LIN {X 0,Y 474.649,Z 278.987,A -85,B 0,C 180,E1 -7371.485,E2 -7371.485} C_VEL
LIN {X 0,Y 474.743,Z 278.967,A -85,B 0,C 180,E1 -7374.052,E2 -7374.052} C_VEL
LIN {X 0,Y 474.863,Z 278.959,A -85,B 0,C 180,E1 -7377.455,E2 -7377.455} C_VEL
LIN {X 0,Y 474.863,Z 278.956,A -85,B 0,C 180,E1 -7380,E2 -7380} C_VEL
LIN {X 0,Y 474.868,Z 278.952,A -85,B 0,C 180,E1 -7382.545,E2 -7382.545} C_VEL
LIN {X 0,Y 474.745,Z 278.969,A -85,B 0,C 180,E1 -7385.948,E2 -7385.948} C_VEL
LIN {X 0,Y 474.696,Z 278.976,A -85,B 0,C 180,E1 -7388.514,E2 -7388.514} C_VEL
LIN {X 0,Y 474.691,Z 278.977,A -85,B 0,C 180,E1 -7391.963,E2 -7391.963} C_VEL
LIN {X 0,Y 474.667,Z 278.98,A -85,B 0,C 180,E1 -7395.767,E2 -7395.767} C_VEL
LIN {X 0,Y 474.65,Z 278.981,A -85,B 0,C 180,E1 -7399.011,E2 -7399.011} C_VEL
LIN {X 0,Y 474.576,Z 278.987,A -85,B 0,C 180,E1 -7401.73,E2 -7401.73} C_VEL
LIN {X 0,Y 474.618,Z 278.988,A -85,B 0,C 180,E1 -7404.495,E2 -7404.495} C_VEL
LIN {X 0,Y 474.663,Z 278.974,A -85,B 0,C 180,E1 -7407.333,E2 -7407.333} C_VEL
LIN {X 0,Y 474.594,Z 278.989,A -85,B 0,C 180,E1 -7410.231,E2 -7410.231} C_VEL
LIN {X 0,Y 474.605,Z 278.991,A -85,B 0,C 180,E1 -7413.223,E2 -7413.223} C_VEL
LIN {X 0,Y 474.58,Z 278.992,A -85,B 0,C 180,E1 -7416.324,E2 -7416.324} C_VEL
LIN {X 0,Y 474.61,Z 278.985,A -85,B 0,C 180,E1 -7419.647,E2 -7419.647} C_VEL
LIN {X 0,Y 474.617,Z 278.987,A -85,B 0,C 180,E1 -7422.237,E2 -7422.237} C_VEL
LIN {X 0,Y 474.611,Z 278.989,A -85,B 0,C 180,E1 -7425.299,E2 -7425.299} C_VEL
LIN {X 0,Y 474.615,Z 278.989,A -85,B 0,C 180,E1 -7428.215,E2 -7428.215} C_VEL
LIN {X 0,Y 474.639,Z 278.988,A -85,B 0,C 180,E1 -7430.455,E2 -7430.455} C_VEL
LIN {X 0,Y 474.585,Z 278.99,A -85,B 0,C 180,E1 -7433.677,E2 -7433.677} C_VEL
LIN {X 0,Y 474.622,Z 278.988,A -85,B 0,C 180,E1 -7436.779,E2 -7436.779} C_VEL
LIN {X 0,Y 474.602,Z 278.991,A -85,B 0,C 180,E1 -7439.771,E2 -7439.771} C_VEL
LIN {X 0,Y 474.73,Z 279.016,A -85,B 0,C 180,E1 -7443.278,E2 -7443.278} C_VEL
LIN {X 0,Y 477.872,Z 293.523,A -85,B 0,C 180,E1 -7445.987,E2 -7445.987} C_VEL
LIN {X 0,Y 478.08,Z 295.472,A -85,B 0,C 180,E1 -7446.3,E2 -7446.3} C_VEL
LIN {X 0,Y 482.601,Z 314.925,A -85,B 0,C 180,E1 -7446.847,E2 -7446.847} C_VEL
LIN {X 0,Y 482.526,Z 323.889,A -85,B 0,C 180,E1 -7446.986,E2 -7446.986} C_VEL
LIN {X 0,Y 481.947,Z 329.738,A -85,B 0,C 180,E1 -7447.049,E2 -7447.049} C_VEL
LIN {X 0,Y 476.326,Z 348.794,A -85,B 0,C 180,E1 -7447.066,E2 -7447.066} C_VEL
LIN {X 0,Y 475.676,Z 354.65,A -85,B 0,C 180,E1 -7447.126,E2 -7447.126} C_VEL
LIN {X 0,Y 474.379,Z 460.534,A -85,B 0,C 180,E1 -7448.781,E2 -7448.781} C_VEL
LIN {X 0,Y 473.901,Z 476.474,A -85,B 0,C 180,E1 -7449.21,E2 -7449.21} C_VEL
LIN {X 0,Y 473.386,Z 491.287,A -85,B 0,C 180,E1 -7449.792,E2 -7449.792} C_VEL
LIN {X 0,Y 472.545,Z 506.177,A -85,B 0,C 180,E1 -7450.563,E2 -7450.563} C_VEL
LIN {X 0,Y 471.802,Z 519.434,A -85,B 0,C 180,E1 -7451.434,E2 -7451.434} C_VEL
LIN {X 0,Y 470.897,Z 532.905,A -85,B 0,C 180,E1 -7452.521,E2 -7452.521} C_VEL
LIN {X 0,Y 470.038,Z 545.12,A -85,B 0,C 180,E1 -7453.719,E2 -7453.719} C_VEL
LIN {X 0,Y 469.245,Z 556.242,A -85,B 0,C 180,E1 -7455.028,E2 -7455.028} C_VEL
LIN {X 0,Y 468.519,Z 567.044,A -85,B 0,C 180,E1 -7456.556,E2 -7456.556} C_VEL
LIN {X 0,Y 467.971,Z 576.004,A -85,B 0,C 180,E1 -7458.083,E2 -7458.083} C_VEL
LIN {X 0,Y 467.459,Z 583.431,A -85,B 0,C 180,E1 -7459.606,E2 -7459.606} C_VEL
LIN {X 0,Y 467.131,Z 590.372,A -85,B 0,C 180,E1 -7461.347,E2 -7461.347} C_VEL
LIN {X 0,Y 466.908,Z 595.827,A -85,B 0,C 180,E1 -7463.084,E2 -7463.084} C_VEL
LIN {X 0,Y 466.75,Z 599.946,A -85,B 0,C 180,E1 -7464.817,E2 -7464.817} C_VEL
LIN {X 0,Y 466.743,Z 602.841,A -85,B 0,C 180,E1 -7466.547,E2 -7466.547} C_VEL
LIN {X 0,Y 466.632,Z 604.587,A -85,B 0,C 180,E1 -7468.274,E2 -7468.274} C_VEL
LIN {X 0,Y 466.597,Z 605.198,A -85,B 0,C 180,E1 -7470,E2 -7470} C_VEL
LIN {X 0,Y 466.633,Z 604.639,A -85,B 0,C 180,E1 -7471.726,E2 -7471.726} C_VEL
LIN {X 0,Y 466.725,Z 602.963,A -85,B 0,C 180,E1 -7473.453,E2 -7473.453} C_VEL
LIN {X 0,Y 466.747,Z 600.134,A -85,B 0,C 180,E1 -7475.183,E2 -7475.183} C_VEL
LIN {X 0,Y 466.906,Z 596.079,A -85,B 0,C 180,E1 -7476.916,E2 -7476.916} C_VEL
LIN {X 0,Y 467.127,Z 590.703,A -85,B 0,C 180,E1 -7478.653,E2 -7478.653} C_VEL
LIN {X 0,Y 467.424,Z 583.853,A -85,B 0,C 180,E1 -7480.394,E2 -7480.394} C_VEL
LIN {X 0,Y 467.931,Z 576.479,A -85,B 0,C 180,E1 -7481.918,E2 -7481.918} C_VEL
LIN {X 0,Y 468.466,Z 567.599,A -85,B 0,C 180,E1 -7483.446,E2 -7483.446} C_VEL
LIN {X 0,Y 469.101,Z 558.541,A -85,B 0,C 180,E1 -7484.755,E2 -7484.755} C_VEL
LIN {X 0,Y 469.852,Z 547.854,A -85,B 0,C 180,E1 -7486.064,E2 -7486.064} C_VEL
LIN {X 0,Y 470.679,Z 536.593,A -85,B 0,C 180,E1 -7487.224,E2 -7487.224} C_VEL
LIN {X 0,Y 471.575,Z 523.439,A -85,B 0,C 180,E1 -7488.35,E2 -7488.35} C_VEL
LIN {X 0,Y 472.393,Z 509.372,A -85,B 0,C 180,E1 -7489.33,E2 -7489.33} C_VEL
LIN {X 0,Y 473.145,Z 496.078,A -85,B 0,C 180,E1 -7490.069,E2 -7490.069} C_VEL
LIN {X 0,Y 473.737,Z 481.419,A -85,B 0,C 180,E1 -7490.704,E2 -7490.704} C_VEL
LIN {X 0,Y 474.199,Z 466.913,A -85,B 0,C 180,E1 -7491.161,E2 -7491.161} C_VEL
LIN {X 0,Y 474.561,Z 450.968,A -85,B 0,C 180,E1 -7491.479,E2 -7491.479} C_VEL
LIN {X 0,Y 476.07,Z 316.361,A -85,B 0,C 180,E1 -7493.562,E2 -7493.562} C_VEL
LIN {X 0,Y 471.893,Z 297.931,A -85,B 0,C 180,E1 -7494.086,E2 -7494.086} C_VEL
LIN {X 0,Y 471.101,Z 295.407,A -85,B 0,C 180,E1 -7494.183,E2 -7494.183} C_VEL
LIN {X 0,Y 468.063,Z 281.748,A -85,B 0,C 180,E1 -7496.772,E2 -7496.772} C_VEL
LIN {X 0,Y 467.662,Z 279.86,A -85,B 0,C 180,E1 -7497.161,E2 -7497.161} C_VEL
LIN {X 0,Y 467.567,Z 279.869,A -85,B 0,C 180,E1 -7500.733,E2 -7500.733} C_VEL
LIN {X 0,Y 467.584,Z 279.868,A -85,B 0,C 180,E1 -7503.787,E2 -7503.787} C_VEL
LIN {X 0,Y 467.546,Z 279.872,A -85,B 0,C 180,E1 -7507.186,E2 -7507.186} C_VEL
LIN {X 0,Y 467.57,Z 279.861,A -85,B 0,C 180,E1 -7510.264,E2 -7510.264} C_VEL
LIN {X 0,Y 467.582,Z 279.865,A -85,B 0,C 180,E1 -7512.566,E2 -7512.566} C_VEL
LIN {X 0,Y 467.56,Z 279.87,A -85,B 0,C 180,E1 -7515.052,E2 -7515.052} C_VEL
LIN {X 0,Y 467.566,Z 279.857,A -85,B 0,C 180,E1 -7518.596,E2 -7518.596} C_VEL
LIN {X 0,Y 467.557,Z 279.862,A -85,B 0,C 180,E1 -7521.955,E2 -7521.955} C_VEL
LIN {X 0,Y 467.55,Z 279.87,A -85,B 0,C 180,E1 -7525.166,E2 -7525.166} C_VEL
LIN {X 0,Y 467.569,Z 279.859,A -85,B 0,C 180,E1 -7528.259,E2 -7528.259} C_VEL
LIN {X 0,Y 467.564,Z 279.868,A -85,B 0,C 180,E1 -7531.249,E2 -7531.249} C_VEL
LIN {X 0,Y 467.578,Z 279.861,A -85,B 0,C 180,E1 -7534.158,E2 -7534.158} C_VEL
LIN {X 0,Y 467.564,Z 279.87,A -85,B 0,C 180,E1 -7536.995,E2 -7536.995} C_VEL
LIN {X 0,Y 467.61,Z 279.859,A -85,B 0,C 180,E1 -7539.776,E2 -7539.776} C_VEL
LIN {X 0,Y 467.584,Z 279.862,A -85,B 0,C 180,E1 -7542.506,E2 -7542.506} C_VEL
LIN {X 0,Y 467.589,Z 279.863,A -85,B 0,C 180,E1 -7545.196,E2 -7545.196} C_VEL
LIN {X 0,Y 467.643,Z 279.854,A -85,B 0,C 180,E1 -7547.854,E2 -7547.854} C_VEL
LIN {X 0,Y 467.654,Z 279.852,A -85,B 0,C 180,E1 -7551.357,E2 -7551.357} C_VEL
LIN {X 0,Y 467.711,Z 279.846,A -85,B 0,C 180,E1 -7553.962,E2 -7553.962} C_VEL
LIN {X 0,Y 467.834,Z 279.832,A -85,B 0,C 180,E1 -7557.417,E2 -7557.417} C_VEL
LIN {X 0,Y 467.862,Z 279.825,A -85,B 0,C 180,E1 -7560,E2 -7560} C_VEL
LIN {X 0,Y 467.805,Z 279.842,A -85,B 0,C 180,E1 -7562.583,E2 -7562.583} C_VEL
LIN {X 0,Y 467.708,Z 279.847,A -85,B 0,C 180,E1 -7566.038,E2 -7566.038} C_VEL
LIN {X 0,Y 467.644,Z 279.856,A -85,B 0,C 180,E1 -7568.643,E2 -7568.643} C_VEL
LIN {X 0,Y 467.642,Z 279.859,A -85,B 0,C 180,E1 -7572.146,E2 -7572.146} C_VEL
LIN {X 0,Y 467.625,Z 279.859,A -85,B 0,C 180,E1 -7575.695,E2 -7575.695} C_VEL
LIN {X 0,Y 467.608,Z 279.86,A -85,B 0,C 180,E1 -7579.308,E2 -7579.308} C_VEL
LIN {X 0,Y 467.519,Z 279.873,A -85,B 0,C 180,E1 -7582.074,E2 -7582.074} C_VEL
LIN {X 0,Y 467.542,Z 279.868,A -85,B 0,C 180,E1 -7584.891,E2 -7584.891} C_VEL
LIN {X 0,Y 467.567,Z 279.867,A -85,B 0,C 180,E1 -7587.772,E2 -7587.772} C_VEL
LIN {X 0,Y 467.556,Z 279.866,A -85,B 0,C 180,E1 -7591.045,E2 -7591.045} C_VEL
LIN {X 0,Y 467.565,Z 279.87,A -85,B 0,C 180,E1 -7594.24,E2 -7594.24} C_VEL
LIN {X 0,Y 467.505,Z 279.871,A -85,B 0,C 180,E1 -7597.181,E2 -7597.181} C_VEL
LIN {X 0,Y 467.549,Z 279.86,A -85,B 0,C 180,E1 -7600.267,E2 -7600.267} C_VEL
LIN {X 0,Y 467.535,Z 279.871,A -85,B 0,C 180,E1 -7602.566,E2 -7602.566} C_VEL
LIN {X 0,Y 467.557,Z 279.866,A -85,B 0,C 180,E1 -7605.053,E2 -7605.053} C_VEL
LIN {X 0,Y 467.553,Z 279.867,A -85,B 0,C 180,E1 -7608.727,E2 -7608.727} C_VEL
LIN {X 0,Y 467.537,Z 279.873,A -85,B 0,C 180,E1 -7611.954,E2 -7611.954} C_VEL
LIN {X 0,Y 467.557,Z 279.869,A -85,B 0,C 180,E1 -7615.168,E2 -7615.168} C_VEL
LIN {X 0,Y 467.579,Z 279.866,A -85,B 0,C 180,E1 -7618.261,E2 -7618.261} C_VEL
LIN {X 0,Y 467.599,Z 280.003,A -85,B 0,C 180,E1 -7619.613,E2 -7619.613} C_VEL
LIN {X 0,Y 471.381,Z 295.697,A -85,B 0,C 180,E1 -7622.298,E2 -7622.298} C_VEL
LIN {X 0,Y 472.191,Z 299.776,A -85,B 0,C 180,E1 -7622.968,E2 -7622.968} C_VEL
LIN {X 0,Y 471.286,Z 317.488,A -85,B 0,C 180,E1 -7625.594,E2 -7625.594} C_VEL
LIN {X 0,Y 471.159,Z 319.301,A -85,B 0,C 180,E1 -7625.859,E2 -7625.859} C_VEL
LIN {X 0,Y 475.892,Z 344.166,A -85,B 0,C 180,E1 -7626.52,E2 -7626.52} C_VEL
LIN {X 0,Y 474.194,Z 484.995,A -85,B 0,C 180,E1 -7628.709,E2 -7628.709} C_VEL
LIN {X 0,Y 473.747,Z 500.567,A -85,B 0,C 180,E1 -7629.115,E2 -7629.115} C_VEL
LIN {X 0,Y 473.071,Z 515.83,A -85,B 0,C 180,E1 -7629.693,E2 -7629.693} C_VEL
LIN {X 0,Y 472.272,Z 530.564,A -85,B 0,C 180,E1 -7630.438,E2 -7630.438} C_VEL
LIN {X 0,Y 471.482,Z 544.074,A -85,B 0,C 180,E1 -7631.308,E2 -7631.308} C_VEL
LIN {X 0,Y 470.612,Z 556.533,A -85,B 0,C 180,E1 -7632.286,E2 -7632.286} C_VEL
LIN {X 0,Y 469.742,Z 569.21,A -85,B 0,C 180,E1 -7633.485,E2 -7633.485} C_VEL
LIN {X 0,Y 468.905,Z 580.728,A -85,B 0,C 180,E1 -7634.794,E2 -7634.794} C_VEL
LIN {X 0,Y 468.32,Z 590.429,A -85,B 0,C 180,E1 -7636.107,E2 -7636.107} C_VEL
LIN {X 0,Y 467.666,Z 599.96,A -85,B 0,C 180,E1 -7637.636,E2 -7637.636} C_VEL
LIN {X 0,Y 467.366,Z 607.901,A -85,B 0,C 180,E1 -7639.166,E2 -7639.166} C_VEL
LIN {X 0,Y 466.985,Z 615.314,A -85,B 0,C 180,E1 -7640.908,E2 -7640.908} C_VEL
LIN {X 0,Y 466.815,Z 621.199,A -85,B 0,C 180,E1 -7642.648,E2 -7642.648} C_VEL
LIN {X 0,Y 466.705,Z 624.696,A -85,B 0,C 180,E1 -7643.949,E2 -7643.949} C_VEL
LIN {X 0,Y 466.614,Z 628.23,A -85,B 0,C 180,E1 -7645.681,E2 -7645.681} C_VEL
LIN {X 0,Y 466.654,Z 630.558,A -85,B 0,C 180,E1 -7647.41,E2 -7647.41} C_VEL
LIN {X 0,Y 466.616,Z 631.728,A -85,B 0,C 180,E1 -7649.137,E2 -7649.137} C_VEL
LIN {X 0,Y 466.616,Z 631.727,A -85,B 0,C 180,E1 -7650.863,E2 -7650.863} C_VEL
LIN {X 0,Y 466.654,Z 630.554,A -85,B 0,C 180,E1 -7652.589,E2 -7652.589} C_VEL
LIN {X 0,Y 466.614,Z 628.226,A -85,B 0,C 180,E1 -7654.319,E2 -7654.319} C_VEL
LIN {X 0,Y 466.698,Z 624.696,A -85,B 0,C 180,E1 -7656.051,E2 -7656.051} C_VEL
LIN {X 0,Y 466.828,Z 619.874,A -85,B 0,C 180,E1 -7657.787,E2 -7657.787} C_VEL
LIN {X 0,Y 467.028,Z 613.628,A -85,B 0,C 180,E1 -7659.528,E2 -7659.528} C_VEL
LIN {X 0,Y 467.483,Z 605.789,A -85,B 0,C 180,E1 -7661.27,E2 -7661.27} C_VEL
LIN {X 0,Y 467.892,Z 597.359,A -85,B 0,C 180,E1 -7662.815,E2 -7662.815} C_VEL
LIN {X 0,Y 468.523,Z 587.409,A -85,B 0,C 180,E1 -7664.33,E2 -7664.33} C_VEL
LIN {X 0,Y 469.194,Z 577.139,A -85,B 0,C 180,E1 -7665.641,E2 -7665.641} C_VEL
LIN {X 0,Y 470.109,Z 564.507,A -85,B 0,C 180,E1 -7666.989,E2 -7666.989} C_VEL
LIN {X 0,Y 470.963,Z 551.302,A -85,B 0,C 180,E1 -7668.15,E2 -7668.15} C_VEL
LIN {X 0,Y 471.842,Z 537.66,A -85,B 0,C 180,E1 -7669.128,E2 -7669.128} C_VEL
LIN {X 0,Y 472.656,Z 523.536,A -85,B 0,C 180,E1 -7669.941,E2 -7669.941} C_VEL
LIN {X 0,Y 473.412,Z 508.346,A -85,B 0,C 180,E1 -7670.614,E2 -7670.614} C_VEL
LIN {X 0,Y 473.982,Z 493.113,A -85,B 0,C 180,E1 -7671.102,E2 -7671.102} C_VEL
LIN {X 0,Y 474.324,Z 477.219,A -85,B 0,C 180,E1 -7671.427,E2 -7671.427} C_VEL
LIN {X 0,Y 475.906,Z 344.039,A -85,B 0,C 180,E1 -7673.48,E2 -7673.48} C_VEL
LIN {X 0,Y 471.162,Z 319.279,A -85,B 0,C 180,E1 -7674.141,E2 -7674.141} C_VEL
LIN {X 0,Y 472.218,Z 301.593,A -85,B 0,C 180,E1 -7676.75,E2 -7676.75} C_VEL
LIN {X 0,Y 471.957,Z 298.284,A -85,B 0,C 180,E1 -7677.269,E2 -7677.269} C_VEL
LIN {X 0,Y 468.654,Z 284.135,A -85,B 0,C 180,E1 -7679.66,E2 -7679.66} C_VEL
LIN {X 0,Y 467.577,Z 279.866,A -85,B 0,C 180,E1 -7680.42,E2 -7680.42} C_VEL
LIN {X 0,Y 467.579,Z 279.867,A -85,B 0,C 180,E1 -7683.788,E2 -7683.788} C_VEL
LIN {X 0,Y 467.506,Z 279.874,A -85,B 0,C 180,E1 -7686.963,E2 -7686.963} C_VEL
LIN {X 0,Y 467.554,Z 279.872,A -85,B 0,C 180,E1 -7689.95,E2 -7689.95} C_VEL
LIN {X 0,Y 467.517,Z 279.874,A -85,B 0,C 180,E1 -7692.567,E2 -7692.567} C_VEL
LIN {X 0,Y 467.557,Z 279.866,A -85,B 0,C 180,E1 -7695.052,E2 -7695.052} C_VEL
LIN {X 0,Y 467.556,Z 279.866,A -85,B 0,C 180,E1 -7698.724,E2 -7698.724} C_VEL
LIN {X 0,Y 467.531,Z 279.873,A -85,B 0,C 180,E1 -7701.952,E2 -7701.952} C_VEL
LIN {X 0,Y 467.54,Z 279.867,A -85,B 0,C 180,E1 -7705.165,E2 -7705.165} C_VEL
LIN {X 0,Y 467.567,Z 279.866,A -85,B 0,C 180,E1 -7708.259,E2 -7708.259} C_VEL
LIN {X 0,Y 467.541,Z 279.869,A -85,B 0,C 180,E1 -7711.248,E2 -7711.248} C_VEL
LIN {X 0,Y 467.551,Z 279.867,A -85,B 0,C 180,E1 -7714.404,E2 -7714.404} C_VEL
LIN {X 0,Y 467.56,Z 279.865,A -85,B 0,C 180,E1 -7716.995,E2 -7716.995} C_VEL
LIN {X 0,Y 467.608,Z 279.855,A -85,B 0,C 180,E1 -7719.777,E2 -7719.777} C_VEL
LIN {X 0,Y 467.576,Z 279.858,A -85,B 0,C 180,E1 -7722.506,E2 -7722.506} C_VEL
LIN {X 0,Y 467.584,Z 279.865,A -85,B 0,C 180,E1 -7725.196,E2 -7725.196} C_VEL
LIN {X 0,Y 467.633,Z 279.842,A -85,B 0,C 180,E1 -7727.854,E2 -7727.854} C_VEL
LIN {X 0,Y 467.617,Z 279.86,A -85,B 0,C 180,E1 -7731.356,E2 -7731.356} C_VEL
LIN {X 0,Y 467.707,Z 279.844,A -85,B 0,C 180,E1 -7733.962,E2 -7733.962} C_VEL
LIN {X 0,Y 467.804,Z 279.839,A -85,B 0,C 180,E1 -7737.417,E2 -7737.417} C_VEL
LIN {X 0,Y 467.833,Z 279.832,A -85,B 0,C 180,E1 -7740,E2 -7740} C_VEL
LIN {X 0,Y 467.809,Z 279.831,A -85,B 0,C 180,E1 -7742.583,E2 -7742.583} C_VEL
LIN {X 0,Y 467.71,Z 279.844,A -85,B 0,C 180,E1 -7746.038,E2 -7746.038} C_VEL
LIN {X 0,Y 467.654,Z 279.854,A -85,B 0,C 180,E1 -7748.643,E2 -7748.643} C_VEL
LIN {X 0,Y 467.643,Z 279.854,A -85,B 0,C 180,E1 -7752.146,E2 -7752.146} C_VEL
LIN {X 0,Y 467.637,Z 279.856,A -85,B 0,C 180,E1 -7755.885,E2 -7755.885} C_VEL
LIN {X 0,Y 467.609,Z 279.853,A -85,B 0,C 180,E1 -7759.308,E2 -7759.308} C_VEL
LIN {X 0,Y 467.522,Z 279.865,A -85,B 0,C 180,E1 -7762.075,E2 -7762.075} C_VEL
LIN {X 0,Y 467.559,Z 279.871,A -85,B 0,C 180,E1 -7764.89,E2 -7764.89} C_VEL
LIN {X 0,Y 467.605,Z 279.851,A -85,B 0,C 180,E1 -7767.77,E2 -7767.77} C_VEL
LIN {X 0,Y 467.557,Z 279.87,A -85,B 0,C 180,E1 -7771.045,E2 -7771.045} C_VEL
LIN {X 0,Y 467.568,Z 279.865,A -85,B 0,C 180,E1 -7774.241,E2 -7774.241} C_VEL
LIN {X 0,Y 467.539,Z 279.869,A -85,B 0,C 180,E1 -7777.187,E2 -7777.187} C_VEL
LIN {X 0,Y 467.567,Z 279.864,A -85,B 0,C 180,E1 -7780.266,E2 -7780.266} C_VEL
LIN {X 0,Y 467.58,Z 279.866,A -85,B 0,C 180,E1 -7782.568,E2 -7782.568} C_VEL
LIN {X 0,Y 467.56,Z 279.87,A -85,B 0,C 180,E1 -7785.053,E2 -7785.053} C_VEL
LIN {X 0,Y 467.584,Z 279.864,A -85,B 0,C 180,E1 -7787.441,E2 -7787.441} C_VEL
LIN {X 0,Y 467.577,Z 279.864,A -85,B 0,C 180,E1 -7790.856,E2 -7790.856} C_VEL
LIN {X 0,Y 467.555,Z 279.867,A -85,B 0,C 180,E1 -7794.262,E2 -7794.262} C_VEL
LIN {X 0,Y 467.576,Z 279.867,A -85,B 0,C 180,E1 -7797.322,E2 -7797.322} C_VEL
LIN {X 0,Y 467.567,Z 279.868,A -85,B 0,C 180,E1 -7800.669,E2 -7800.669} C_VEL
LIN {X 0,Y 467.682,Z 279.982,A -85,B 0,C 180,E1 -7802.98,E2 -7802.98} C_VEL
LIN {X 0,Y 470.958,Z 294.754,A -85,B 0,C 180,E1 -7805.787,E2 -7805.787} C_VEL
LIN {X 0,Y 471.113,Z 295.593,A -85,B 0,C 180,E1 -7805.925,E2 -7805.925} C_VEL
LIN {X 0,Y 474.546,Z 308.99,A -85,B 0,C 180,E1 -7806.33,E2 -7806.33} C_VEL
LIN {X 0,Y 476.068,Z 316.337,A -85,B 0,C 180,E1 -7806.53,E2 -7806.53} C_VEL
LIN {X 0,Y 475.676,Z 354.65,A -85,B 0,C 180,E1 -7807.126,E2 -7807.126} C_VEL
LIN {X 0,Y 475.049,Z 360.502,A -85,B 0,C 180,E1 -7807.188,E2 -7807.188} C_VEL
LIN {X 0,Y 469.472,Z 379.568,A -85,B 0,C 180,E1 -7807.209,E2 -7807.209} C_VEL
LIN {X 0,Y 468.768,Z 385.426,A -85,B 0,C 180,E1 -7807.268,E2 -7807.268} C_VEL
LIN {X 0,Y 467.778,Z 460.757,A -85,B 0,C 180,E1 -7808.467,E2 -7808.467} C_VEL
LIN {X 0,Y 467.292,Z 476.353,A -85,B 0,C 180,E1 -7808.889,E2 -7808.889} C_VEL
LIN {X 0,Y 466.791,Z 490.68,A -85,B 0,C 180,E1 -7809.455,E2 -7809.455} C_VEL
LIN {X 0,Y 465.971,Z 504.495,A -85,B 0,C 180,E1 -7810.163,E2 -7810.163} C_VEL
LIN {X 0,Y 465.187,Z 518.081,A -85,B 0,C 180,E1 -7811.046,E2 -7811.046} C_VEL
LIN {X 0,Y 464.3,Z 530.573,A -85,B 0,C 180,E1 -7812.037,E2 -7812.037} C_VEL
LIN {X 0,Y 463.387,Z 543.219,A -85,B 0,C 180,E1 -7813.252,E2 -7813.252} C_VEL
LIN {X 0,Y 462.512,Z 554.681,A -85,B 0,C 180,E1 -7814.579,E2 -7814.579} C_VEL
LIN {X 0,Y 461.803,Z 564.324,A -85,B 0,C 180,E1 -7815.907,E2 -7815.907} C_VEL
LIN {X 0,Y 461.027,Z 573.959,A -85,B 0,C 180,E1 -7817.488,E2 -7817.488} C_VEL
LIN {X 0,Y 460.604,Z 581.637,A -85,B 0,C 180,E1 -7819.005,E2 -7819.005} C_VEL
LIN {X 0,Y 460.146,Z 588.979,A -85,B 0,C 180,E1 -7820.772,E2 -7820.772} C_VEL
LIN {X 0,Y 459.899,Z 594.802,A -85,B 0,C 180,E1 -7822.537,E2 -7822.537} C_VEL
LIN {X 0,Y 459.779,Z 598.249,A -85,B 0,C 180,E1 -7823.858,E2 -7823.858} C_VEL
LIN {X 0,Y 459.592,Z 601.747,A -85,B 0,C 180,E1 -7825.615,E2 -7825.615} C_VEL
LIN {X 0,Y 459.601,Z 604.058,A -85,B 0,C 180,E1 -7827.371,E2 -7827.371} C_VEL
LIN {X 0,Y 459.52,Z 605.243,A -85,B 0,C 180,E1 -7829.124,E2 -7829.124} C_VEL
LIN {X 0,Y 459.521,Z 605.26,A -85,B 0,C 180,E1 -7830.876,E2 -7830.876} C_VEL
LIN {X 0,Y 459.6,Z 604.144,A -85,B 0,C 180,E1 -7832.629,E2 -7832.629} C_VEL
LIN {X 0,Y 459.591,Z 601.9,A -85,B 0,C 180,E1 -7834.385,E2 -7834.385} C_VEL
LIN {X 0,Y 459.772,Z 598.466,A -85,B 0,C 180,E1 -7836.142,E2 -7836.142} C_VEL
LIN {X 0,Y 459.962,Z 593.766,A -85,B 0,C 180,E1 -7837.904,E2 -7837.904} C_VEL
LIN {X 0,Y 460.235,Z 587.676,A -85,B 0,C 180,E1 -7839.67,E2 -7839.67} C_VEL
LIN {X 0,Y 460.796,Z 580.002,A -85,B 0,C 180,E1 -7841.436,E2 -7841.436} C_VEL
LIN {X 0,Y 461.258,Z 571.926,A -85,B 0,C 180,E1 -7842.969,E2 -7842.969} C_VEL
LIN {X 0,Y 461.992,Z 561.966,A -85,B 0,C 180,E1 -7844.537,E2 -7844.537} C_VEL
LIN {X 0,Y 462.72,Z 551.857,A -85,B 0,C 180,E1 -7845.866,E2 -7845.866} C_VEL
LIN {X 0,Y 463.578,Z 540.956,A -85,B 0,C 180,E1 -7847.073,E2 -7847.073} C_VEL
LIN {X 0,Y 464.396,Z 529.032,A -85,B 0,C 180,E1 -7848.187,E2 -7848.187} C_VEL
LIN {X 0,Y 465.352,Z 516.2,A -85,B 0,C 180,E1 -7849.176,E2 -7849.176} C_VEL
LIN {X 0,Y 466.143,Z 502.129,A -85,B 0,C 180,E1 -7850.059,E2 -7850.059} C_VEL
LIN {X 0,Y 466.92,Z 487.101,A -85,B 0,C 180,E1 -7850.79,E2 -7850.79} C_VEL
LIN {X 0,Y 467.438,Z 472.322,A -85,B 0,C 180,E1 -7851.325,E2 -7851.325} C_VEL
LIN {X 0,Y 467.809,Z 457.776,A -85,B 0,C 180,E1 -7851.683,E2 -7851.683} C_VEL
LIN {X 0,Y 468.791,Z 380.02,A -85,B 0,C 180,E1 -7852.911,E2 -7852.911} C_VEL
LIN {X 0,Y 469.453,Z 316.407,A -85,B 0,C 180,E1 -7853.917,E2 -7853.917} C_VEL
LIN {X 0,Y 465.461,Z 299.692,A -85,B 0,C 180,E1 -7854.414,E2 -7854.414} C_VEL
LIN {X 0,Y 463.967,Z 295.631,A -85,B 0,C 180,E1 -7854.577,E2 -7854.577} C_VEL
LIN {X 0,Y 460.595,Z 280.738,A -85,B 0,C 180,E1 -7857.47,E2 -7857.47} C_VEL
LIN {X 0,Y 460.508,Z 280.749,A -85,B 0,C 180,E1 -7860.239,E2 -7860.239} C_VEL
LIN {X 0,Y 460.527,Z 280.751,A -85,B 0,C 180,E1 -7863.324,E2 -7863.324} C_VEL
LIN {X 0,Y 460.475,Z 280.753,A -85,B 0,C 180,E1 -7866.528,E2 -7866.528} C_VEL
LIN {X 0,Y 460.537,Z 280.746,A -85,B 0,C 180,E1 -7868.896,E2 -7868.896} C_VEL
LIN {X 0,Y 460.518,Z 280.744,A -85,B 0,C 180,E1 -7872.18,E2 -7872.18} C_VEL
LIN {X 0,Y 460.507,Z 280.75,A -85,B 0,C 180,E1 -7875.41,E2 -7875.41} C_VEL
LIN {X 0,Y 460.52,Z 280.738,A -85,B 0,C 180,E1 -7878.987,E2 -7878.987} C_VEL
LIN {X 0,Y 460.509,Z 280.747,A -85,B 0,C 180,E1 -7881.265,E2 -7881.265} C_VEL
LIN {X 0,Y 460.5,Z 280.74,A -85,B 0,C 180,E1 -7884.553,E2 -7884.553} C_VEL
LIN {X 0,Y 460.516,Z 280.739,A -85,B 0,C 180,E1 -7887.714,E2 -7887.714} C_VEL
LIN {X 0,Y 460.528,Z 280.736,A -85,B 0,C 180,E1 -7890.768,E2 -7890.768} C_VEL
LIN {X 0,Y 460.532,Z 280.739,A -85,B 0,C 180,E1 -7893.733,E2 -7893.733} C_VEL
LIN {X 0,Y 460.533,Z 280.744,A -85,B 0,C 180,E1 -7896.623,E2 -7896.623} C_VEL
LIN {X 0,Y 460.539,Z 280.742,A -85,B 0,C 180,E1 -7899.452,E2 -7899.452} C_VEL
LIN {X 0,Y 460.535,Z 280.738,A -85,B 0,C 180,E1 -7902.229,E2 -7902.229} C_VEL
LIN {X 0,Y 460.55,Z 280.743,A -85,B 0,C 180,E1 -7904.964,E2 -7904.964} C_VEL
LIN {X 0,Y 460.595,Z 280.736,A -85,B 0,C 180,E1 -7908.559,E2 -7908.559} C_VEL
LIN {X 0,Y 460.604,Z 280.732,A -85,B 0,C 180,E1 -7911.223,E2 -7911.223} C_VEL
LIN {X 0,Y 460.677,Z 280.722,A -85,B 0,C 180,E1 -7913.87,E2 -7913.87} C_VEL
LIN {X 0,Y 460.775,Z 280.711,A -85,B 0,C 180,E1 -7917.377,E2 -7917.377} C_VEL
LIN {X 0,Y 460.833,Z 280.7,A -85,B 0,C 180,E1 -7920,E2 -7920} C_VEL
LIN {X 0,Y 460.749,Z 280.72,A -85,B 0,C 180,E1 -7922.623,E2 -7922.623} C_VEL
LIN {X 0,Y 460.674,Z 280.724,A -85,B 0,C 180,E1 -7926.13,E2 -7926.13} C_VEL
LIN {X 0,Y 460.593,Z 280.733,A -85,B 0,C 180,E1 -7928.777,E2 -7928.777} C_VEL
LIN {X 0,Y 460.584,Z 280.739,A -85,B 0,C 180,E1 -7932.435,E2 -7932.435} C_VEL
LIN {X 0,Y 460.567,Z 280.74,A -85,B 0,C 180,E1 -7935.988,E2 -7935.988} C_VEL
LIN {X 0,Y 460.554,Z 280.739,A -85,B 0,C 180,E1 -7939.616,E2 -7939.616} C_VEL
LIN {X 0,Y 460.496,Z 280.749,A -85,B 0,C 180,E1 -7942.429,E2 -7942.429} C_VEL
LIN {X 0,Y 460.512,Z 280.744,A -85,B 0,C 180,E1 -7945.791,E2 -7945.791} C_VEL
LIN {X 0,Y 460.513,Z 280.75,A -85,B 0,C 180,E1 -7948.235,E2 -7948.235} C_VEL
LIN {X 0,Y 460.51,Z 280.744,A -85,B 0,C 180,E1 -7951.283,E2 -7951.283} C_VEL
LIN {X 0,Y 460.509,Z 280.748,A -85,B 0,C 180,E1 -7954.504,E2 -7954.504} C_VEL
LIN {X 0,Y 460.473,Z 280.749,A -85,B 0,C 180,E1 -7957.626,E2 -7957.626} C_VEL
LIN {X 0,Y 460.509,Z 280.735,A -85,B 0,C 180,E1 -7961.014,E2 -7961.014} C_VEL
LIN {X 0,Y 460.504,Z 280.747,A -85,B 0,C 180,E1 -7964.59,E2 -7964.59} C_VEL
LIN {X 0,Y 460.467,Z 280.754,A -85,B 0,C 180,E1 -7967.814,E2 -7967.814} C_VEL
LIN {X 0,Y 460.503,Z 280.748,A -85,B 0,C 180,E1 -7970.136,E2 -7970.136} C_VEL
LIN {X 0,Y 460.46,Z 280.752,A -85,B 0,C 180,E1 -7973.47,E2 -7973.47} C_VEL
LIN {X 0,Y 460.523,Z 280.746,A -85,B 0,C 180,E1 -7976.676,E2 -7976.676} C_VEL
LIN {X 0,Y 460.545,Z 280.79,A -85,B 0,C 180,E1 -7979.256,E2 -7979.256} C_VEL
LIN {X 0,Y 464.356,Z 296.633,A -85,B 0,C 180,E1 -7982.02,E2 -7982.02} C_VEL
LIN {X 0,Y 465.393,Z 302.525,A -85,B 0,C 180,E1 -7982.995,E2 -7982.995} C_VEL
LIN {X 0,Y 464.398,Z 319.103,A -85,B 0,C 180,E1 -7985.486,E2 -7985.486} C_VEL
LIN {X 0,Y 469.38,Z 344.927,A -85,B 0,C 180,E1 -7986.189,E2 -7986.189} C_VEL
LIN {X 0,Y 467.596,Z 484.807,A -85,B 0,C 180,E1 -7988.394,E2 -7988.394} C_VEL
LIN {X 0,Y 467.093,Z 500.372,A -85,B 0,C 180,E1 -7988.803,E2 -7988.803} C_VEL
LIN {X 0,Y 466.404,Z 514.627,A -85,B 0,C 180,E1 -7989.345,E2 -7989.345} C_VEL
LIN {X 0,Y 465.698,Z 528.373,A -85,B 0,C 180,E1 -7990.036,E2 -7990.036} C_VEL
LIN {X 0,Y 464.781,Z 542.286,A -85,B 0,C 180,E1 -7990.914,E2 -7990.914} C_VEL
LIN {X 0,Y 463.854,Z 555.035,A -85,B 0,C 180,E1 -7991.905,E2 -7991.905} C_VEL
LIN {X 0,Y 463.001,Z 566.73,A -85,B 0,C 180,E1 -7992.997,E2 -7992.997} C_VEL
LIN {X 0,Y 462.119,Z 578.733,A -85,B 0,C 180,E1 -7994.339,E2 -7994.339} C_VEL
LIN {X 0,Y 461.431,Z 588.731,A -85,B 0,C 180,E1 -7995.671,E2 -7995.671} C_VEL
LIN {X 0,Y 460.769,Z 598.761,A -85,B 0,C 180,E1 -7997.268,E2 -7997.268} C_VEL
LIN {X 0,Y 460.422,Z 606.682,A -85,B 0,C 180,E1 -7998.778,E2 -7998.778} C_VEL
LIN {X 0,Y 459.956,Z 613.429,A -85,B 0,C 180,E1 -8000.324,E2 -8000.324} C_VEL
LIN {X 0,Y 459.769,Z 619.668,A -85,B 0,C 180,E1 -8002.093,E2 -8002.093} C_VEL
LIN {X 0,Y 459.617,Z 624.493,A -85,B 0,C 180,E1 -8003.856,E2 -8003.856} C_VEL
LIN {X 0,Y 459.53,Z 628.028,A -85,B 0,C 180,E1 -8005.614,E2 -8005.614} C_VEL
LIN {X 0,Y 459.574,Z 630.356,A -85,B 0,C 180,E1 -8007.371,E2 -8007.371} C_VEL
LIN {X 0,Y 459.519,Z 631.525,A -85,B 0,C 180,E1 -8009.124,E2 -8009.124} C_VEL
LIN {X 0,Y 459.519,Z 631.524,A -85,B 0,C 180,E1 -8010.876,E2 -8010.876} C_VEL
LIN {X 0,Y 459.574,Z 630.351,A -85,B 0,C 180,E1 -8012.629,E2 -8012.629} C_VEL
LIN {X 0,Y 459.53,Z 628.022,A -85,B 0,C 180,E1 -8014.386,E2 -8014.386} C_VEL
LIN {X 0,Y 459.617,Z 624.492,A -85,B 0,C 180,E1 -8016.144,E2 -8016.144} C_VEL
LIN {X 0,Y 459.769,Z 619.67,A -85,B 0,C 180,E1 -8017.907,E2 -8017.907} C_VEL
LIN {X 0,Y 459.956,Z 613.422,A -85,B 0,C 180,E1 -8019.676,E2 -8019.676} C_VEL
LIN {X 0,Y 460.407,Z 606.671,A -85,B 0,C 180,E1 -8021.223,E2 -8021.223} C_VEL
LIN {X 0,Y 460.789,Z 598.755,A -85,B 0,C 180,E1 -8022.732,E2 -8022.732} C_VEL
LIN {X 0,Y 461.449,Z 588.724,A -85,B 0,C 180,E1 -8024.329,E2 -8024.329} C_VEL
LIN {X 0,Y 462.135,Z 578.723,A -85,B 0,C 180,E1 -8025.66,E2 -8025.66} C_VEL
LIN {X 0,Y 462.942,Z 568.334,A -85,B 0,C 180,E1 -8026.835,E2 -8026.835} C_VEL
LIN {X 0,Y 463.776,Z 556.321,A -85,B 0,C 180,E1 -8027.984,E2 -8027.984} C_VEL
LIN {X 0,Y 464.681,Z 543.844,A -85,B 0,C 180,E1 -8028.975,E2 -8028.975} C_VEL
LIN {X 0,Y 465.617,Z 530.324,A -85,B 0,C 180,E1 -8029.853,E2 -8029.853} C_VEL
LIN {X 0,Y 466.358,Z 516.338,A -85,B 0,C 180,E1 -8030.578,E2 -8030.578} C_VEL
LIN {X 0,Y 467.055,Z 501.191,A -85,B 0,C 180,E1 -8031.17,E2 -8031.17} C_VEL
LIN {X 0,Y 467.55,Z 486.044,A -85,B 0,C 180,E1 -8031.58,E2 -8031.58} C_VEL
LIN {X 0,Y 469.206,Z 359.073,A -85,B 0,C 180,E1 -8033.586,E2 -8033.586} C_VEL
LIN {X 0,Y 469.302,Z 344.153,A -85,B 0,C 180,E1 -8033.825,E2 -8033.825} C_VEL
LIN {X 0,Y 464.413,Z 318.949,A -85,B 0,C 180,E1 -8034.533,E2 -8034.533} C_VEL
LIN {X 0,Y 465.393,Z 302.491,A -85,B 0,C 180,E1 -8037.005,E2 -8037.005} C_VEL
LIN {X 0,Y 464.368,Z 296.608,A -85,B 0,C 180,E1 -8037.98,E2 -8037.98} C_VEL
LIN {X 0,Y 460.937,Z 282.339,A -85,B 0,C 180,E1 -8040.461,E2 -8040.461} C_VEL
LIN {X 0,Y 460.544,Z 280.741,A -85,B 0,C 180,E1 -8040.776,E2 -8040.776} C_VEL
LIN {X 0,Y 460.523,Z 280.744,A -85,B 0,C 180,E1 -8043.324,E2 -8043.324} C_VEL
LIN {X 0,Y 460.46,Z 280.754,A -85,B 0,C 180,E1 -8046.53,E2 -8046.53} C_VEL
LIN {X 0,Y 460.503,Z 280.75,A -85,B 0,C 180,E1 -8049.864,E2 -8049.864} C_VEL
LIN {X 0,Y 460.458,Z 280.751,A -85,B 0,C 180,E1 -8052.893,E2 -8052.893} C_VEL
LIN {X 0,Y 460.496,Z 280.751,A -85,B 0,C 180,E1 -8055.831,E2 -8055.831} C_VEL
LIN {X 0,Y 460.509,Z 280.744,A -85,B 0,C 180,E1 -8058.986,E2 -8058.986} C_VEL
LIN {X 0,Y 460.473,Z 280.75,A -85,B 0,C 180,E1 -8062.374,E2 -8062.374} C_VEL
LIN {X 0,Y 460.523,Z 280.745,A -85,B 0,C 180,E1 -8065.622,E2 -8065.622} C_VEL
LIN {X 0,Y 460.528,Z 280.741,A -85,B 0,C 180,E1 -8068.744,E2 -8068.744} C_VEL
LIN {X 0,Y 460.507,Z 280.75,A -85,B 0,C 180,E1 -8071.764,E2 -8071.764} C_VEL
LIN {X 0,Y 460.5,Z 280.745,A -85,B 0,C 180,E1 -8074.702,E2 -8074.702} C_VEL
LIN {X 0,Y 460.495,Z 280.751,A -85,B 0,C 180,E1 -8077.571,E2 -8077.571} C_VEL
LIN {X 0,Y 460.554,Z 280.727,A -85,B 0,C 180,E1 -8080.384,E2 -8080.384} C_VEL
LIN {X 0,Y 460.593,Z 280.735,A -85,B 0,C 180,E1 -8084.059,E2 -8084.059} C_VEL
LIN {X 0,Y 460.589,Z 280.722,A -85,B 0,C 180,E1 -8087.665,E2 -8087.665} C_VEL
LIN {X 0,Y 460.571,Z 280.736,A -85,B 0,C 180,E1 -8091.223,E2 -8091.223} C_VEL
LIN {X 0,Y 460.673,Z 280.721,A -85,B 0,C 180,E1 -8093.87,E2 -8093.87} C_VEL
LIN {X 0,Y 460.748,Z 280.719,A -85,B 0,C 180,E1 -8097.377,E2 -8097.377} C_VEL
LIN {X 0,Y 460.782,Z 280.711,A -85,B 0,C 180,E1 -8100,E2 -8100} C_VEL
LIN {X 0,Y 460.754,Z 280.71,A -85,B 0,C 180,E1 -8102.623,E2 -8102.623} C_VEL
LIN {X 0,Y 460.677,Z 280.72,A -85,B 0,C 180,E1 -8106.13,E2 -8106.13} C_VEL
LIN {X 0,Y 460.604,Z 280.733,A -85,B 0,C 180,E1 -8108.777,E2 -8108.777} C_VEL
LIN {X 0,Y 460.585,Z 280.734,A -85,B 0,C 180,E1 -8112.435,E2 -8112.435} C_VEL
LIN {X 0,Y 460.589,Z 280.733,A -85,B 0,C 180,E1 -8115.998,E2 -8115.998} C_VEL
LIN {X 0,Y 460.555,Z 280.727,A -85,B 0,C 180,E1 -8119.616,E2 -8119.616} C_VEL
LIN {X 0,Y 460.498,Z 280.74,A -85,B 0,C 180,E1 -8122.429,E2 -8122.429} C_VEL
LIN {X 0,Y 460.536,Z 280.736,A -85,B 0,C 180,E1 -8125.797,E2 -8125.797} C_VEL
LIN {X 0,Y 460.539,Z 280.731,A -85,B 0,C 180,E1 -8128.234,E2 -8128.234} C_VEL
LIN {X 0,Y 460.511,Z 280.745,A -85,B 0,C 180,E1 -8131.283,E2 -8131.283} C_VEL
LIN {X 0,Y 460.514,Z 280.745,A -85,B 0,C 180,E1 -8134.505,E2 -8134.505} C_VEL
LIN {X 0,Y 460.493,Z 280.744,A -85,B 0,C 180,E1 -8137.624,E2 -8137.624} C_VEL
LIN {X 0,Y 460.531,Z 280.74,A -85,B 0,C 180,E1 -8140.27,E2 -8140.27} C_VEL
LIN {X 0,Y 460.49,Z 280.748,A -85,B 0,C 180,E1 -8143.377,E2 -8143.377} C_VEL
LIN {X 0,Y 460.493,Z 280.751,A -85,B 0,C 180,E1 -8146.625,E2 -8146.625} C_VEL
LIN {X 0,Y 460.537,Z 280.742,A -85,B 0,C 180,E1 -8149.732,E2 -8149.732} C_VEL
LIN {X 0,Y 460.495,Z 280.75,A -85,B 0,C 180,E1 -8152.525,E2 -8152.525} C_VEL
LIN {X 0,Y 460.534,Z 280.743,A -85,B 0,C 180,E1 -8155.624,E2 -8155.624} C_VEL
LIN {X 0,Y 460.535,Z 280.743,A -85,B 0,C 180,E1 -8158.745,E2 -8158.745} C_VEL
LIN {X 0,Y 460.579,Z 280.734,A -85,B 0,C 180,E1 -8162.255,E2 -8162.255} C_VEL
LIN {X 0,Y 460.631,Z 280.748,A -85,B 0,C 180,E1 -8162.637,E2 -8162.637} C_VEL
LIN {X 0,Y 463.94,Z 295.643,A -85,B 0,C 180,E1 -8165.515,E2 -8165.515} C_VEL
LIN {X 0,Y 466.224,Z 302.441,A -85,B 0,C 180,E1 -8165.767,E2 -8165.767} C_VEL
LIN {X 0,Y 469.582,Z 317.442,A -85,B 0,C 180,E1 -8166.2,E2 -8166.2} C_VEL
LIN {X 0,Y 468.768,Z 385.426,A -85,B 0,C 180,E1 -8167.268,E2 -8167.268} C_VEL
LIN {X 0,Y 468.084,Z 391.278,A -85,B 0,C 180,E1 -8167.328,E2 -8167.328} C_VEL
LIN {X 0,Y 462.579,Z 410.348,A -85,B 0,C 180,E1 -8167.355,E2 -8167.355} C_VEL
LIN {X 0,Y 461.878,Z 416.201,A -85,B 0,C 180,E1 -8167.415,E2 -8167.415} C_VEL
LIN {X 0,Y 461.192,Z 460.98,A -85,B 0,C 180,E1 -8168.143,E2 -8168.143} C_VEL
LIN {X 0,Y 460.689,Z 476.767,A -85,B 0,C 180,E1 -8168.58,E2 -8168.58} C_VEL
LIN {X 0,Y 460.152,Z 491.141,A -85,B 0,C 180,E1 -8169.157,E2 -8169.157} C_VEL
LIN {X 0,Y 459.302,Z 504.706,A -85,B 0,C 180,E1 -8169.863,E2 -8169.863} C_VEL
LIN {X 0,Y 458.468,Z 518.29,A -85,B 0,C 180,E1 -8170.757,E2 -8170.757} C_VEL
LIN {X 0,Y 457.52,Z 530.782,A -85,B 0,C 180,E1 -8171.762,E2 -8171.762} C_VEL
LIN {X 0,Y 456.584,Z 543.426,A -85,B 0,C 180,E1 -8172.995,E2 -8172.995} C_VEL
LIN {X 0,Y 455.651,Z 554.888,A -85,B 0,C 180,E1 -8174.341,E2 -8174.341} C_VEL
LIN {X 0,Y 454.899,Z 564.531,A -85,B 0,C 180,E1 -8175.689,E2 -8175.689} C_VEL
LIN {X 0,Y 454.157,Z 573.328,A -85,B 0,C 180,E1 -8177.139,E2 -8177.139} C_VEL
LIN {X 0,Y 453.628,Z 581.843,A -85,B 0,C 180,E1 -8178.834,E2 -8178.834} C_VEL
LIN {X 0,Y 453.12,Z 589.184,A -85,B 0,C 180,E1 -8180.627,E2 -8180.627} C_VEL
LIN {X 0,Y 452.836,Z 595.007,A -85,B 0,C 180,E1 -8182.42,E2 -8182.42} C_VEL
LIN {X 0,Y 452.71,Z 598.453,A -85,B 0,C 180,E1 -8183.762,E2 -8183.762} C_VEL
LIN {X 0,Y 452.511,Z 601.951,A -85,B 0,C 180,E1 -8185.546,E2 -8185.546} C_VEL
LIN {X 0,Y 452.526,Z 604.261,A -85,B 0,C 180,E1 -8187.33,E2 -8187.33} C_VEL
LIN {X 0,Y 452.428,Z 605.446,A -85,B 0,C 180,E1 -8189.11,E2 -8189.11} C_VEL
LIN {X 0,Y 452.428,Z 605.463,A -85,B 0,C 180,E1 -8190.89,E2 -8190.89} C_VEL
LIN {X 0,Y 452.525,Z 604.346,A -85,B 0,C 180,E1 -8192.67,E2 -8192.67} C_VEL
LIN {X 0,Y 452.509,Z 602.102,A -85,B 0,C 180,E1 -8194.454,E2 -8194.454} C_VEL
LIN {X 0,Y 452.685,Z 598.668,A -85,B 0,C 180,E1 -8196.239,E2 -8196.239} C_VEL
LIN {X 0,Y 452.911,Z 593.968,A -85,B 0,C 180,E1 -8198.028,E2 -8198.028} C_VEL
LIN {X 0,Y 453.216,Z 587.878,A -85,B 0,C 180,E1 -8199.821,E2 -8199.821} C_VEL
LIN {X 0,Y 453.783,Z 580.205,A -85,B 0,C 180,E1 -8201.615,E2 -8201.615} C_VEL
LIN {X 0,Y 454.286,Z 572.342,A -85,B 0,C 180,E1 -8203.132,E2 -8203.132} C_VEL
LIN {X 0,Y 455.091,Z 562.167,A -85,B 0,C 180,E1 -8204.762,E2 -8204.762} C_VEL
LIN {X 0,Y 455.859,Z 552.057,A -85,B 0,C 180,E1 -8206.111,E2 -8206.111} C_VEL
LIN {X 0,Y 456.716,Z 541.757,A -85,B 0,C 180,E1 -8207.272,E2 -8207.272} C_VEL
LIN {X 0,Y 457.644,Z 529.23,A -85,B 0,C 180,E1 -8208.465,E2 -8208.465} C_VEL
LIN {X 0,Y 458.647,Z 516.397,A -85,B 0,C 180,E1 -8209.468,E2 -8209.468} C_VEL
LIN {X 0,Y 459.376,Z 504.306,A -85,B 0,C 180,E1 -8210.251,E2 -8210.251} C_VEL
LIN {X 0,Y 460.119,Z 491.665,A -85,B 0,C 180,E1 -8210.912,E2 -8210.912} C_VEL
LIN {X 0,Y 460.711,Z 476.947,A -85,B 0,C 180,E1 -8211.505,E2 -8211.505} C_VEL
LIN {X 0,Y 461.128,Z 462.082,A -85,B 0,C 180,E1 -8211.925,E2 -8211.925} C_VEL
LIN {X 0,Y 461.837,Z 421.293,A -85,B 0,C 180,E1 -8212.596,E2 -8212.596} C_VEL
LIN {X 0,Y 463.079,Z 318.391,A -85,B 0,C 180,E1 -8214.237,E2 -8214.237} C_VEL
LIN {X 0,Y 459.227,Z 301.922,A -85,B 0,C 180,E1 -8214.733,E2 -8214.733} C_VEL
LIN {X 0,Y 456.81,Z 295.856,A -85,B 0,C 180,E1 -8214.986,E2 -8214.986} C_VEL
LIN {X 0,Y 453.548,Z 281.616,A -85,B 0,C 180,E1 -8217.827,E2 -8217.827} C_VEL
LIN {X 0,Y 453.474,Z 281.626,A -85,B 0,C 180,E1 -8220.759,E2 -8220.759} C_VEL
LIN {X 0,Y 453.475,Z 281.625,A -85,B 0,C 180,E1 -8223.912,E2 -8223.912} C_VEL
LIN {X 0,Y 453.45,Z 281.627,A -85,B 0,C 180,E1 -8227.189,E2 -8227.189} C_VEL
LIN {X 0,Y 453.482,Z 281.623,A -85,B 0,C 180,E1 -8229.449,E2 -8229.449} C_VEL
LIN {X 0,Y 453.471,Z 281.624,A -85,B 0,C 180,E1 -8231.934,E2 -8231.934} C_VEL
LIN {X 0,Y 453.477,Z 281.626,A -85,B 0,C 180,E1 -8235.47,E2 -8235.47} C_VEL
LIN {X 0,Y 453.456,Z 281.613,A -85,B 0,C 180,E1 -8238.207,E2 -8238.207} C_VEL
LIN {X 0,Y 453.461,Z 281.625,A -85,B 0,C 180,E1 -8240.797,E2 -8240.797} C_VEL
LIN {X 0,Y 453.445,Z 281.618,A -85,B 0,C 180,E1 -8243.916,E2 -8243.916} C_VEL
LIN {X 0,Y 453.465,Z 281.623,A -85,B 0,C 180,E1 -8247.15,E2 -8247.15} C_VEL
LIN {X 0,Y 453.464,Z 281.612,A -85,B 0,C 180,E1 -8250.267,E2 -8250.267} C_VEL
LIN {X 0,Y 453.522,Z 281.614,A -85,B 0,C 180,E1 -8252.297,E2 -8252.297} C_VEL
LIN {X 0,Y 453.482,Z 281.624,A -85,B 0,C 180,E1 -8255.264,E2 -8255.264} C_VEL
LIN {X 0,Y 453.47,Z 281.619,A -85,B 0,C 180,E1 -8258.415,E2 -8258.415} C_VEL
LIN {X 0,Y 453.512,Z 281.619,A -85,B 0,C 180,E1 -8261.008,E2 -8261.008} C_VEL
LIN {X 0,Y 453.558,Z 281.609,A -85,B 0,C 180,E1 -8263.879,E2 -8263.879} C_VEL
LIN {X 0,Y 453.552,Z 281.61,A -85,B 0,C 180,E1 -8267.471,E2 -8267.471} C_VEL
LIN {X 0,Y 453.57,Z 281.608,A -85,B 0,C 180,E1 -8271.086,E2 -8271.086} C_VEL
LIN {X 0,Y 453.645,Z 281.598,A -85,B 0,C 180,E1 -8273.774,E2 -8273.774} C_VEL
LIN {X 0,Y 453.719,Z 281.59,A -85,B 0,C 180,E1 -8277.336,E2 -8277.336} C_VEL
LIN {X 0,Y 453.803,Z 281.576,A -85,B 0,C 180,E1 -8280,E2 -8280} C_VEL
LIN {X 0,Y 453.696,Z 281.598,A -85,B 0,C 180,E1 -8282.663,E2 -8282.663} C_VEL
LIN {X 0,Y 453.642,Z 281.601,A -85,B 0,C 180,E1 -8286.226,E2 -8286.226} C_VEL
LIN {X 0,Y 453.559,Z 281.609,A -85,B 0,C 180,E1 -8288.914,E2 -8288.914} C_VEL
LIN {X 0,Y 453.552,Z 281.613,A -85,B 0,C 180,E1 -8292.529,E2 -8292.529} C_VEL
LIN {X 0,Y 453.526,Z 281.62,A -85,B 0,C 180,E1 -8296.197,E2 -8296.197} C_VEL
LIN {X 0,Y 453.505,Z 281.618,A -85,B 0,C 180,E1 -8299.039,E2 -8299.039} C_VEL
LIN {X 0,Y 453.464,Z 281.622,A -85,B 0,C 180,E1 -8301.837,E2 -8301.837} C_VEL
LIN {X 0,Y 453.453,Z 281.624,A -85,B 0,C 180,E1 -8304.738,E2 -8304.738} C_VEL
LIN {X 0,Y 453.488,Z 281.622,A -85,B 0,C 180,E1 -8307.952,E2 -8307.952} C_VEL
LIN {X 0,Y 453.465,Z 281.623,A -85,B 0,C 180,E1 -8310.76,E2 -8310.76} C_VEL
LIN {X 0,Y 453.455,Z 281.622,A -85,B 0,C 180,E1 -8313.914,E2 -8313.914} C_VEL
LIN {X 0,Y 453.425,Z 281.625,A -85,B 0,C 180,E1 -8317.192,E2 -8317.192} C_VEL
LIN {X 0,Y 453.462,Z 281.612,A -85,B 0,C 180,E1 -8320.612,E2 -8320.612} C_VEL
LIN {X 0,Y 453.451,Z 281.627,A -85,B 0,C 180,E1 -8324.223,E2 -8324.223} C_VEL
LIN {X 0,Y 453.414,Z 281.628,A -85,B 0,C 180,E1 -8327.001,E2 -8327.001} C_VEL
LIN {X 0,Y 453.464,Z 281.623,A -85,B 0,C 180,E1 -8329.413,E2 -8329.413} C_VEL
LIN {X 0,Y 453.433,Z 281.625,A -85,B 0,C 180,E1 -8332.81,E2 -8332.81} C_VEL
LIN {X 0,Y 453.471,Z 281.626,A -85,B 0,C 180,E1 -8336.088,E2 -8336.088} C_VEL
LIN {X 0,Y 453.521,Z 281.688,A -85,B 0,C 180,E1 -8338.907,E2 -8338.907} C_VEL
LIN {X 0,Y 457.479,Z 298.007,A -85,B 0,C 180,E1 -8341.811,E2 -8341.811} C_VEL
LIN {X 0,Y 458.576,Z 303.428,A -85,B 0,C 180,E1 -8342.734,E2 -8342.734} C_VEL
LIN {X 0,Y 457.668,Z 318.906,A -85,B 0,C 180,E1 -8345.102,E2 -8345.102} C_VEL
LIN {X 0,Y 462.811,Z 345.144,A -85,B 0,C 180,E1 -8345.837,E2 -8345.837} C_VEL
LIN {X 0,Y 461.312,Z 464.422,A -85,B 0,C 180,E1 -8347.731,E2 -8347.731} C_VEL
LIN {X 0,Y 460.95,Z 487.078,A -85,B 0,C 180,E1 -8348.125,E2 -8348.125} C_VEL
LIN {X 0,Y 460.374,Z 502.405,A -85,B 0,C 180,E1 -8348.56,E2 -8348.56} C_VEL
LIN {X 0,Y 459.667,Z 516.672,A -85,B 0,C 180,E1 -8349.134,E2 -8349.134} C_VEL
LIN {X 0,Y 458.87,Z 530.165,A -85,B 0,C 180,E1 -8349.843,E2 -8349.843} C_VEL
LIN {X 0,Y 457.927,Z 543.671,A -85,B 0,C 180,E1 -8350.734,E2 -8350.734} C_VEL
LIN {X 0,Y 456.954,Z 556.129,A -85,B 0,C 180,E1 -8351.738,E2 -8351.738} C_VEL
LIN {X 0,Y 456.028,Z 568.805,A -85,B 0,C 180,E1 -8352.974,E2 -8352.974} C_VEL
LIN {X 0,Y 455.087,Z 580.322,A -85,B 0,C 180,E1 -8354.321,E2 -8354.321} C_VEL
LIN {X 0,Y 454.381,Z 590.022,A -85,B 0,C 180,E1 -8355.672,E2 -8355.672} C_VEL
LIN {X 0,Y 453.694,Z 599.549,A -85,B 0,C 180,E1 -8357.248,E2 -8357.248} C_VEL
LIN {X 0,Y 453.326,Z 607.494,A -85,B 0,C 180,E1 -8358.826,E2 -8358.826} C_VEL
LIN {X 0,Y 452.839,Z 614.906,A -85,B 0,C 180,E1 -8360.622,E2 -8360.622} C_VEL
LIN {X 0,Y 452.654,Z 620.792,A -85,B 0,C 180,E1 -8362.417,E2 -8362.417} C_VEL
LIN {X 0,Y 452.542,Z 624.29,A -85,B 0,C 180,E1 -8363.759,E2 -8363.759} C_VEL
LIN {X 0,Y 452.448,Z 627.825,A -85,B 0,C 180,E1 -8365.546,E2 -8365.546} C_VEL
LIN {X 0,Y 452.496,Z 630.153,A -85,B 0,C 180,E1 -8367.329,E2 -8367.329} C_VEL
LIN {X 0,Y 452.426,Z 631.322,A -85,B 0,C 180,E1 -8369.11,E2 -8369.11} C_VEL
LIN {X 0,Y 452.426,Z 631.321,A -85,B 0,C 180,E1 -8370.89,E2 -8370.89} C_VEL
LIN {X 0,Y 452.496,Z 630.148,A -85,B 0,C 180,E1 -8372.671,E2 -8372.671} C_VEL
LIN {X 0,Y 452.448,Z 627.819,A -85,B 0,C 180,E1 -8374.454,E2 -8374.454} C_VEL
LIN {X 0,Y 452.512,Z 624.179,A -85,B 0,C 180,E1 -8376.287,E2 -8376.287} C_VEL
LIN {X 0,Y 452.692,Z 619.465,A -85,B 0,C 180,E1 -8378.032,E2 -8378.032} C_VEL
LIN {X 0,Y 452.895,Z 613.217,A -85,B 0,C 180,E1 -8379.828,E2 -8379.828} C_VEL
LIN {X 0,Y 453.354,Z 606.465,A -85,B 0,C 180,E1 -8381.399,E2 -8381.399} C_VEL
LIN {X 0,Y 453.807,Z 598.549,A -85,B 0,C 180,E1 -8382.931,E2 -8382.931} C_VEL
LIN {X 0,Y 454.396,Z 590.012,A -85,B 0,C 180,E1 -8384.327,E2 -8384.327} C_VEL
LIN {X 0,Y 455.101,Z 580.308,A -85,B 0,C 180,E1 -8385.679,E2 -8385.679} C_VEL
LIN {X 0,Y 456.028,Z 568.792,A -85,B 0,C 180,E1 -8387.026,E2 -8387.026} C_VEL
LIN {X 0,Y 456.937,Z 556.112,A -85,B 0,C 180,E1 -8388.263,E2 -8388.263} C_VEL
LIN {X 0,Y 457.926,Z 543.636,A -85,B 0,C 180,E1 -8389.266,E2 -8389.266} C_VEL
LIN {X 0,Y 458.901,Z 530.115,A -85,B 0,C 180,E1 -8390.156,E2 -8390.156} C_VEL
LIN {X 0,Y 459.67,Z 516.647,A -85,B 0,C 180,E1 -8390.865,E2 -8390.865} C_VEL
LIN {X 0,Y 460.396,Z 501.773,A -85,B 0,C 180,E1 -8391.461,E2 -8391.461} C_VEL
LIN {X 0,Y 460.96,Z 485.83,A -85,B 0,C 180,E1 -8391.904,E2 -8391.904} C_VEL
LIN {X 0,Y 462.658,Z 363.053,A -85,B 0,C 180,E1 -8393.871,E2 -8393.871} C_VEL
LIN {X 0,Y 462.818,Z 345.192,A -85,B 0,C 180,E1 -8394.159,E2 -8394.159} C_VEL
LIN {X 0,Y 457.657,Z 318.739,A -85,B 0,C 180,E1 -8394.919,E2 -8394.919} C_VEL
LIN {X 0,Y 458.574,Z 303.395,A -85,B 0,C 180,E1 -8397.265,E2 -8397.265} C_VEL
LIN {X 0,Y 455.975,Z 291.56,A -85,B 0,C 180,E1 -8399.311,E2 -8399.311} C_VEL
LIN {X 0,Y 453.508,Z 281.618,A -85,B 0,C 180,E1 -8401.124,E2 -8401.124} C_VEL
LIN {X 0,Y 453.471,Z 281.624,A -85,B 0,C 180,E1 -8403.912,E2 -8403.912} C_VEL
LIN {X 0,Y 453.433,Z 281.628,A -85,B 0,C 180,E1 -8407.19,E2 -8407.19} C_VEL
LIN {X 0,Y 453.463,Z 281.625,A -85,B 0,C 180,E1 -8410.611,E2 -8410.611} C_VEL
LIN {X 0,Y 453.451,Z 281.629,A -85,B 0,C 180,E1 -8414.221,E2 -8414.221} C_VEL
LIN {X 0,Y 453.428,Z 281.626,A -85,B 0,C 180,E1 -8417.001,E2 -8417.001} C_VEL
LIN {X 0,Y 453.462,Z 281.624,A -85,B 0,C 180,E1 -8419.412,E2 -8419.412} C_VEL
LIN {X 0,Y 453.426,Z 281.626,A -85,B 0,C 180,E1 -8422.808,E2 -8422.808} C_VEL
LIN {X 0,Y 453.455,Z 281.625,A -85,B 0,C 180,E1 -8426.086,E2 -8426.086} C_VEL
LIN {X 0,Y 453.465,Z 281.622,A -85,B 0,C 180,E1 -8429.24,E2 -8429.24} C_VEL
LIN {X 0,Y 453.48,Z 281.618,A -85,B 0,C 180,E1 -8432.294,E2 -8432.294} C_VEL
LIN {X 0,Y 453.452,Z 281.625,A -85,B 0,C 180,E1 -8435.262,E2 -8435.262} C_VEL
LIN {X 0,Y 453.469,Z 281.62,A -85,B 0,C 180,E1 -8438.415,E2 -8438.415} C_VEL
LIN {X 0,Y 453.511,Z 281.604,A -85,B 0,C 180,E1 -8441.008,E2 -8441.008} C_VEL
LIN {X 0,Y 453.557,Z 281.614,A -85,B 0,C 180,E1 -8443.879,E2 -8443.879} C_VEL
LIN {X 0,Y 453.552,Z 281.601,A -85,B 0,C 180,E1 -8447.471,E2 -8447.471} C_VEL
LIN {X 0,Y 453.541,Z 281.61,A -85,B 0,C 180,E1 -8451.086,E2 -8451.086} C_VEL
LIN {X 0,Y 453.64,Z 281.598,A -85,B 0,C 180,E1 -8453.774,E2 -8453.774} C_VEL
LIN {X 0,Y 453.695,Z 281.598,A -85,B 0,C 180,E1 -8457.337,E2 -8457.337} C_VEL
LIN {X 0,Y 453.733,Z 281.589,A -85,B 0,C 180,E1 -8460,E2 -8460} C_VEL
LIN {X 0,Y 453.701,Z 281.589,A -85,B 0,C 180,E1 -8462.664,E2 -8462.664} C_VEL
LIN {X 0,Y 453.645,Z 281.596,A -85,B 0,C 180,E1 -8466.226,E2 -8466.226} C_VEL
LIN {X 0,Y 453.57,Z 281.611,A -85,B 0,C 180,E1 -8468.914,E2 -8468.914} C_VEL
LIN {X 0,Y 453.552,Z 281.61,A -85,B 0,C 180,E1 -8472.529,E2 -8472.529} C_VEL
LIN {X 0,Y 453.533,Z 281.612,A -85,B 0,C 180,E1 -8476.196,E2 -8476.196} C_VEL
LIN {X 0,Y 453.506,Z 281.613,A -85,B 0,C 180,E1 -8479.04,E2 -8479.04} C_VEL
LIN {X 0,Y 453.465,Z 281.616,A -85,B 0,C 180,E1 -8481.837,E2 -8481.837} C_VEL
LIN {X 0,Y 453.482,Z 281.623,A -85,B 0,C 180,E1 -8484.736,E2 -8484.736} C_VEL
LIN {X 0,Y 453.519,Z 281.605,A -85,B 0,C 180,E1 -8487.959,E2 -8487.959} C_VEL
LIN {X 0,Y 453.454,Z 281.621,A -85,B 0,C 180,E1 -8491.525,E2 -8491.525} C_VEL
LIN {X 0,Y 453.474,Z 281.624,A -85,B 0,C 180,E1 -8494.777,E2 -8494.777} C_VEL
LIN {X 0,Y 453.455,Z 281.622,A -85,B 0,C 180,E1 -8498.313,E2 -8498.313} C_VEL
LIN {X 0,Y 453.487,Z 281.62,A -85,B 0,C 180,E1 -8500.61,E2 -8500.61} C_VEL
LIN {X 0,Y 453.447,Z 281.626,A -85,B 0,C 180,E1 -8503.245,E2 -8503.245} C_VEL
LIN {X 0,Y 453.458,Z 281.623,A -85,B 0,C 180,E1 -8505.78,E2 -8505.78} C_VEL
LIN {X 0,Y 453.474,Z 281.623,A -85,B 0,C 180,E1 -8508.21,E2 -8508.21} C_VEL
LIN {X 0,Y 453.51,Z 281.616,A -85,B 0,C 180,E1 -8510.791,E2 -8510.791} C_VEL
LIN {X 0,Y 453.45,Z 281.623,A -85,B 0,C 180,E1 -8513.918,E2 -8513.918} C_VEL
LIN {X 0,Y 453.476,Z 281.623,A -85,B 0,C 180,E1 -8517.152,E2 -8517.152} C_VEL
LIN {X 0,Y 453.472,Z 281.626,A -85,B 0,C 180,E1 -8520.269,E2 -8520.269} C_VEL
LIN {X 0,Y 453.553,Z 281.627,A -85,B 0,C 180,E1 -8522.3,E2 -8522.3} C_VEL
LIN {X 0,Y 456.7,Z 295.471,A -85,B 0,C 180,E1 -8525.031,E2 -8525.031} C_VEL
LIN {X 0,Y 456.876,Z 296.253,A -85,B 0,C 180,E1 -8525.128,E2 -8525.128} C_VEL
LIN {X 0,Y 459.831,Z 304.066,A -85,B 0,C 180,E1 -8525.432,E2 -8525.432} C_VEL
LIN {X 0,Y 463.104,Z 318.611,A -85,B 0,C 180,E1 -8525.862,E2 -8525.862} C_VEL
LIN {X 0,Y 461.878,Z 416.201,A -85,B 0,C 180,E1 -8527.415,E2 -8527.415} C_VEL
LIN {X 0,Y 461.164,Z 422.047,A -85,B 0,C 180,E1 -8527.475,E2 -8527.475} C_VEL
LIN {X 0,Y 455.564,Z 441.073,A -85,B 0,C 180,E1 -8527.498,E2 -8527.498} C_VEL
LIN {X 0,Y 454.88,Z 446.918,A -85,B 0,C 180,E1 -8527.56,E2 -8527.56} C_VEL
LIN {X 0,Y 454.479,Z 464.981,A -85,B 0,C 180,E1 -8527.902,E2 -8527.902} C_VEL
LIN {X 0,Y 453.961,Z 480.055,A -85,B 0,C 180,E1 -8528.367,E2 -8528.367} C_VEL
LIN {X 0,Y 453.299,Z 495.027,A -85,B 0,C 180,E1 -8529.019,E2 -8529.019} C_VEL
LIN {X 0,Y 452.406,Z 508.566,A -85,B 0,C 180,E1 -8529.779,E2 -8529.779} C_VEL
LIN {X 0,Y 451.521,Z 521.492,A -85,B 0,C 180,E1 -8530.686,E2 -8530.686} C_VEL
LIN {X 0,Y 450.579,Z 533.53,A -85,B 0,C 180,E1 -8531.706,E2 -8531.706} C_VEL
LIN {X 0,Y 449.581,Z 545.743,A -85,B 0,C 180,E1 -8532.956,E2 -8532.956} C_VEL
LIN {X 0,Y 448.621,Z 556.864,A -85,B 0,C 180,E1 -8534.322,E2 -8534.322} C_VEL
LIN {X 0,Y 447.716,Z 567.665,A -85,B 0,C 180,E1 -8535.918,E2 -8535.918} C_VEL
LIN {X 0,Y 446.982,Z 576.625,A -85,B 0,C 180,E1 -8537.515,E2 -8537.515} C_VEL
LIN {X 0,Y 446.423,Z 584.049,A -85,B 0,C 180,E1 -8539.111,E2 -8539.111} C_VEL
LIN {X 0,Y 446.002,Z 590.988,A -85,B 0,C 180,E1 -8540.934,E2 -8540.934} C_VEL
LIN {X 0,Y 445.722,Z 596.441,A -85,B 0,C 180,E1 -8542.754,E2 -8542.754} C_VEL
LIN {X 0,Y 445.568,Z 600.557,A -85,B 0,C 180,E1 -8544.57,E2 -8544.57} C_VEL
LIN {X 0,Y 445.454,Z 603.452,A -85,B 0,C 180,E1 -8546.382,E2 -8546.382} C_VEL
LIN {X 0,Y 445.377,Z 605.196,A -85,B 0,C 180,E1 -8548.192,E2 -8548.192} C_VEL
LIN {X 0,Y 445.34,Z 605.806,A -85,B 0,C 180,E1 -8550,E2 -8550} C_VEL
LIN {X 0,Y 445.377,Z 605.246,A -85,B 0,C 180,E1 -8551.808,E2 -8551.808} C_VEL
LIN {X 0,Y 445.44,Z 603.57,A -85,B 0,C 180,E1 -8553.618,E2 -8553.618} C_VEL
LIN {X 0,Y 445.563,Z 600.739,A -85,B 0,C 180,E1 -8555.43,E2 -8555.43} C_VEL
LIN {X 0,Y 445.715,Z 596.686,A -85,B 0,C 180,E1 -8557.247,E2 -8557.247} C_VEL
LIN {X 0,Y 445.993,Z 591.31,A -85,B 0,C 180,E1 -8559.066,E2 -8559.066} C_VEL
LIN {X 0,Y 446.403,Z 584.458,A -85,B 0,C 180,E1 -8560.89,E2 -8560.89} C_VEL
LIN {X 0,Y 446.95,Z 577.085,A -85,B 0,C 180,E1 -8562.486,E2 -8562.486} C_VEL
LIN {X 0,Y 447.675,Z 568.202,A -85,B 0,C 180,E1 -8564.083,E2 -8564.083} C_VEL
LIN {X 0,Y 448.442,Z 559.143,A -85,B 0,C 180,E1 -8565.451,E2 -8565.451} C_VEL
LIN {X 0,Y 449.33,Z 548.454,A -85,B 0,C 180,E1 -8566.819,E2 -8566.819} C_VEL
LIN {X 0,Y 450.339,Z 536.882,A -85,B 0,C 180,E1 -8568.059,E2 -8568.059} C_VEL
LIN {X 0,Y 451.282,Z 525.451,A -85,B 0,C 180,E1 -8569.089,E2 -8569.089} C_VEL
LIN {X 0,Y 452.225,Z 511.721,A -85,B 0,C 180,E1 -8570.111,E2 -8570.111} C_VEL
LIN {X 0,Y 453.074,Z 498.509,A -85,B 0,C 180,E1 -8570.901,E2 -8570.901} C_VEL
LIN {X 0,Y 453.869,Z 482.927,A -85,B 0,C 180,E1 -8571.618,E2 -8571.618} C_VEL
LIN {X 0,Y 454.422,Z 467.957,A -85,B 0,C 180,E1 -8572.116,E2 -8572.116} C_VEL
LIN {X 0,Y 454.81,Z 453.617,A -85,B 0,C 180,E1 -8572.425,E2 -8572.425} C_VEL
LIN {X 0,Y 455.753,Z 380.371,A -85,B 0,C 180,E1 -8573.606,E2 -8573.606} C_VEL
LIN {X 0,Y 456.505,Z 318.695,A -85,B 0,C 180,E1 -8574.607,E2 -8574.607} C_VEL
LIN {X 0,Y 453.095,Z 304.527,A -85,B 0,C 180,E1 -8575.049,E2 -8575.049} C_VEL
LIN {X 0,Y 449.633,Z 296.006,A -85,B 0,C 180,E1 -8575.425,E2 -8575.425} C_VEL
LIN {X 0,Y 446.498,Z 282.496,A -85,B 0,C 180,E1 -8578.155,E2 -8578.155} C_VEL
LIN {X 0,Y 446.417,Z 282.505,A -85,B 0,C 180,E1 -8581.774,E2 -8581.774} C_VEL
LIN {X 0,Y 446.427,Z 282.5,A -85,B 0,C 180,E1 -8584.522,E2 -8584.522} C_VEL
LIN {X 0,Y 446.426,Z 282.503,A -85,B 0,C 180,E1 -8588.081,E2 -8588.081} C_VEL
LIN {X 0,Y 446.422,Z 282.497,A -85,B 0,C 180,E1 -8590.917,E2 -8590.917} C_VEL
LIN {X 0,Y 446.394,Z 282.505,A -85,B 0,C 180,E1 -8593.845,E2 -8593.845} C_VEL
LIN {X 0,Y 446.392,Z 282.503,A -85,B 0,C 180,E1 -8596.403,E2 -8596.403} C_VEL
LIN {X 0,Y 446.429,Z 282.499,A -85,B 0,C 180,E1 -8599.8,E2 -8599.8} C_VEL
LIN {X 0,Y 446.394,Z 282.495,A -85,B 0,C 180,E1 -8603.254,E2 -8603.254} C_VEL
LIN {X 0,Y 446.44,Z 282.498,A -85,B 0,C 180,E1 -8606.566,E2 -8606.566} C_VEL
LIN {X 0,Y 446.419,Z 282.489,A -85,B 0,C 180,E1 -8609.979,E2 -8609.979} C_VEL
LIN {X 0,Y 446.454,Z 282.499,A -85,B 0,C 180,E1 -8612.838,E2 -8612.838} C_VEL
LIN {X 0,Y 446.45,Z 282.495,A -85,B 0,C 180,E1 -8615.924,E2 -8615.924} C_VEL
LIN {X 0,Y 446.442,Z 282.496,A -85,B 0,C 180,E1 -8618.772,E2 -8618.772} C_VEL
LIN {X 0,Y 446.439,Z 282.493,A -85,B 0,C 180,E1 -8621.648,E2 -8621.648} C_VEL
LIN {X 0,Y 446.495,Z 282.492,A -85,B 0,C 180,E1 -8624.479,E2 -8624.479} C_VEL
LIN {X 0,Y 446.503,Z 282.488,A -85,B 0,C 180,E1 -8628.193,E2 -8628.193} C_VEL
LIN {X 0,Y 446.518,Z 282.487,A -85,B 0,C 180,E1 -8630.944,E2 -8630.944} C_VEL
LIN {X 0,Y 446.615,Z 282.474,A -85,B 0,C 180,E1 -8633.676,E2 -8633.676} C_VEL
LIN {X 0,Y 446.666,Z 282.469,A -85,B 0,C 180,E1 -8637.294,E2 -8637.294} C_VEL
LIN {X 0,Y 446.773,Z 282.452,A -85,B 0,C 180,E1 -8640,E2 -8640} C_VEL
LIN {X 0,Y 446.646,Z 282.476,A -85,B 0,C 180,E1 -8642.706,E2 -8642.706} C_VEL
LIN {X 0,Y 446.611,Z 282.477,A -85,B 0,C 180,E1 -8646.324,E2 -8646.324} C_VEL
LIN {X 0,Y 446.507,Z 282.486,A -85,B 0,C 180,E1 -8649.056,E2 -8649.056} C_VEL
LIN {X 0,Y 446.51,Z 282.488,A -85,B 0,C 180,E1 -8652.73,E2 -8652.73} C_VEL
LIN {X 0,Y 446.473,Z 282.498,A -85,B 0,C 180,E1 -8656.46,E2 -8656.46} C_VEL
LIN {X 0,Y 446.457,Z 282.495,A -85,B 0,C 180,E1 -8659.304,E2 -8659.304} C_VEL
LIN {X 0,Y 446.405,Z 282.502,A -85,B 0,C 180,E1 -8662.2,E2 -8662.2} C_VEL
LIN {X 0,Y 446.403,Z 282.5,A -85,B 0,C 180,E1 -8665.155,E2 -8665.155} C_VEL
LIN {X 0,Y 446.433,Z 282.504,A -85,B 0,C 180,E1 -8668.182,E2 -8668.182} C_VEL
LIN {X 0,Y 446.404,Z 282.501,A -85,B 0,C 180,E1 -8671.301,E2 -8671.301} C_VEL
LIN {X 0,Y 446.41,Z 282.504,A -85,B 0,C 180,E1 -8674.525,E2 -8674.525} C_VEL
LIN {X 0,Y 446.388,Z 282.509,A -85,B 0,C 180,E1 -8678.077,E2 -8678.077} C_VEL
LIN {X 0,Y 446.398,Z 282.493,A -85,B 0,C 180,E1 -8681.394,E2 -8681.394} C_VEL
LIN {X 0,Y 446.414,Z 282.501,A -85,B 0,C 180,E1 -8684.893,E2 -8684.893} C_VEL
LIN {X 0,Y 446.393,Z 282.504,A -85,B 0,C 180,E1 -8688.606,E2 -8688.606} C_VEL
LIN {X 0,Y 446.394,Z 282.506,A -85,B 0,C 180,E1 -8691.924,E2 -8691.924} C_VEL
LIN {X 0,Y 446.423,Z 282.503,A -85,B 0,C 180,E1 -8695.478,E2 -8695.478} C_VEL
LIN {X 0,Y 446.453,Z 282.63,A -85,B 0,C 180,E1 -8698.551,E2 -8698.551} C_VEL
LIN {X 0,Y 450.108,Z 297.386,A -85,B 0,C 180,E1 -8701.241,E2 -8701.241} C_VEL
LIN {X 0,Y 451.788,Z 305.626,A -85,B 0,C 180,E1 -8702.674,E2 -8702.674} C_VEL
LIN {X 0,Y 450.909,Z 318.659,A -85,B 0,C 180,E1 -8704.697,E2 -8704.697} C_VEL
LIN {X 0,Y 456.362,Z 346.558,A -85,B 0,C 180,E1 -8705.5,E2 -8705.5} C_VEL
LIN {X 0,Y 454.417,Z 484.43,A -85,B 0,C 180,E1 -8707.734,E2 -8707.734} C_VEL
LIN {X 0,Y 453.863,Z 499.983,A -85,B 0,C 180,E1 -8708.154,E2 -8708.154} C_VEL
LIN {X 0,Y 453.082,Z 514.976,A -85,B 0,C 180,E1 -8708.743,E2 -8708.743} C_VEL
LIN {X 0,Y 452.194,Z 529.966,A -85,B 0,C 180,E1 -8709.532,E2 -8709.532} C_VEL
LIN {X 0,Y 451.181,Z 543.471,A -85,B 0,C 180,E1 -8710.434,E2 -8710.434} C_VEL
LIN {X 0,Y 450.08,Z 557.223,A -85,B 0,C 180,E1 -8711.567,E2 -8711.567} C_VEL
LIN {X 0,Y 449.09,Z 569.742,A -85,B 0,C 180,E1 -8712.827,E2 -8712.827} C_VEL
LIN {X 0,Y 448.038,Z 581.891,A -85,B 0,C 180,E1 -8714.301,E2 -8714.301} C_VEL
LIN {X 0,Y 447.22,Z 592.757,A -85,B 0,C 180,E1 -8715.902,E2 -8715.902} C_VEL
LIN {X 0,Y 446.512,Z 602.069,A -85,B 0,C 180,E1 -8717.555,E2 -8717.555} C_VEL
LIN {X 0,Y 446.139,Z 609.32,A -85,B 0,C 180,E1 -8719.104,E2 -8719.104} C_VEL
LIN {X 0,Y 445.709,Z 616.327,A -85,B 0,C 180,E1 -8720.928,E2 -8720.928} C_VEL
LIN {X 0,Y 445.569,Z 621.842,A -85,B 0,C 180,E1 -8722.751,E2 -8722.751} C_VEL
LIN {X 0,Y 445.408,Z 626.01,A -85,B 0,C 180,E1 -8724.568,E2 -8724.568} C_VEL
LIN {X 0,Y 445.336,Z 628.932,A -85,B 0,C 180,E1 -8726.381,E2 -8726.381} C_VEL
LIN {X 0,Y 445.352,Z 630.677,A -85,B 0,C 180,E1 -8728.191,E2 -8728.191} C_VEL
LIN {X 0,Y 445.339,Z 631.274,A -85,B 0,C 180,E1 -8730,E2 -8730} C_VEL
LIN {X 0,Y 445.352,Z 630.674,A -85,B 0,C 180,E1 -8731.809,E2 -8731.809} C_VEL
LIN {X 0,Y 445.336,Z 628.925,A -85,B 0,C 180,E1 -8733.619,E2 -8733.619} C_VEL
LIN {X 0,Y 445.403,Z 626.005,A -85,B 0,C 180,E1 -8735.432,E2 -8735.432} C_VEL
LIN {X 0,Y 445.504,Z 621.84,A -85,B 0,C 180,E1 -8737.25,E2 -8737.25} C_VEL
LIN {X 0,Y 445.709,Z 616.322,A -85,B 0,C 180,E1 -8739.072,E2 -8739.072} C_VEL
LIN {X 0,Y 446.136,Z 609.305,A -85,B 0,C 180,E1 -8740.896,E2 -8740.896} C_VEL
LIN {X 0,Y 446.62,Z 600.571,A -85,B 0,C 180,E1 -8742.726,E2 -8742.726} C_VEL
LIN {X 0,Y 447.339,Z 591.299,A -85,B 0,C 180,E1 -8744.326,E2 -8744.326} C_VEL
LIN {X 0,Y 448.051,Z 581.873,A -85,B 0,C 180,E1 -8745.698,E2 -8745.698} C_VEL
LIN {X 0,Y 449.024,Z 570.714,A -85,B 0,C 180,E1 -8747.061,E2 -8747.061} C_VEL
LIN {X 0,Y 449.971,Z 558.423,A -85,B 0,C 180,E1 -8748.32,E2 -8748.32} C_VEL
LIN {X 0,Y 451.064,Z 544.95,A -85,B 0,C 180,E1 -8749.453,E2 -8749.453} C_VEL
LIN {X 0,Y 452.076,Z 531.725,A -85,B 0,C 180,E1 -8750.355,E2 -8750.355} C_VEL
LIN {X 0,Y 452.925,Z 518.162,A -85,B 0,C 180,E1 -8751.099,E2 -8751.099} C_VEL
LIN {X 0,Y 453.648,Z 503.925,A -85,B 0,C 180,E1 -8751.704,E2 -8751.704} C_VEL
LIN {X 0,Y 454.235,Z 489.044,A -85,B 0,C 180,E1 -8752.156,E2 -8752.156} C_VEL
LIN {X 0,Y 454.649,Z 469.395,A -85,B 0,C 180,E1 -8752.523,E2 -8752.523} C_VEL
LIN {X 0,Y 456.388,Z 347.252,A -85,B 0,C 180,E1 -8754.483,E2 -8754.483} C_VEL
LIN {X 0,Y 450.909,Z 318.665,A -85,B 0,C 180,E1 -8755.297,E2 -8755.297} C_VEL
LIN {X 0,Y 451.787,Z 305.593,A -85,B 0,C 180,E1 -8757.326,E2 -8757.326} C_VEL
LIN {X 0,Y 449.482,Z 294.599,A -85,B 0,C 180,E1 -8759.248,E2 -8759.248} C_VEL
LIN {X 0,Y 446.423,Z 282.498,A -85,B 0,C 180,E1 -8761.473,E2 -8761.473} C_VEL
LIN {X 0,Y 446.423,Z 282.503,A -85,B 0,C 180,E1 -8764.522,E2 -8764.522} C_VEL
LIN {X 0,Y 446.393,Z 282.507,A -85,B 0,C 180,E1 -8768.076,E2 -8768.076} C_VEL
LIN {X 0,Y 446.394,Z 282.505,A -85,B 0,C 180,E1 -8771.393,E2 -8771.393} C_VEL
LIN {X 0,Y 446.414,Z 282.501,A -85,B 0,C 180,E1 -8774.892,E2 -8774.892} C_VEL
LIN {X 0,Y 446.384,Z 282.507,A -85,B 0,C 180,E1 -8777.728,E2 -8777.728} C_VEL
LIN {X 0,Y 446.389,Z 282.503,A -85,B 0,C 180,E1 -8780.967,E2 -8780.967} C_VEL
LIN {X 0,Y 446.4,Z 282.501,A -85,B 0,C 180,E1 -8784.372,E2 -8784.372} C_VEL
LIN {X 0,Y 446.407,Z 282.502,A -85,B 0,C 180,E1 -8787.637,E2 -8787.637} C_VEL
LIN {X 0,Y 446.416,Z 282.498,A -85,B 0,C 180,E1 -8790.788,E2 -8790.788} C_VEL
LIN {X 0,Y 446.424,Z 282.504,A -85,B 0,C 180,E1 -8793.845,E2 -8793.845} C_VEL
LIN {X 0,Y 446.41,Z 282.499,A -85,B 0,C 180,E1 -8796.822,E2 -8796.822} C_VEL
LIN {X 0,Y 446.431,Z 282.492,A -85,B 0,C 180,E1 -8799.737,E2 -8799.737} C_VEL
LIN {X 0,Y 446.438,Z 282.491,A -85,B 0,C 180,E1 -8802.596,E2 -8802.596} C_VEL
LIN {X 0,Y 446.45,Z 282.501,A -85,B 0,C 180,E1 -8805.412,E2 -8805.412} C_VEL
LIN {X 0,Y 446.492,Z 282.471,A -85,B 0,C 180,E1 -8808.192,E2 -8808.192} C_VEL
LIN {X 0,Y 446.492,Z 282.487,A -85,B 0,C 180,E1 -8810.944,E2 -8810.944} C_VEL
LIN {X 0,Y 446.609,Z 282.475,A -85,B 0,C 180,E1 -8813.676,E2 -8813.676} C_VEL
LIN {X 0,Y 446.644,Z 282.477,A -85,B 0,C 180,E1 -8817.294,E2 -8817.294} C_VEL
LIN {X 0,Y 446.684,Z 282.467,A -85,B 0,C 180,E1 -8820,E2 -8820} C_VEL
LIN {X 0,Y 446.651,Z 282.467,A -85,B 0,C 180,E1 -8822.706,E2 -8822.706} C_VEL
LIN {X 0,Y 446.614,Z 282.472,A -85,B 0,C 180,E1 -8826.324,E2 -8826.324} C_VEL
LIN {X 0,Y 446.518,Z 282.491,A -85,B 0,C 180,E1 -8829.056,E2 -8829.056} C_VEL
LIN {X 0,Y 446.51,Z 282.489,A -85,B 0,C 180,E1 -8832.73,E2 -8832.73} C_VEL
LIN {X 0,Y 446.477,Z 282.492,A -85,B 0,C 180,E1 -8836.46,E2 -8836.46} C_VEL
LIN {X 0,Y 446.457,Z 282.486,A -85,B 0,C 180,E1 -8839.304,E2 -8839.304} C_VEL
LIN {X 0,Y 446.406,Z 282.495,A -85,B 0,C 180,E1 -8842.2,E2 -8842.2} C_VEL
LIN {X 0,Y 446.427,Z 282.499,A -85,B 0,C 180,E1 -8845.154,E2 -8845.154} C_VEL
LIN {X 0,Y 446.476,Z 282.482,A -85,B 0,C 180,E1 -8848.179,E2 -8848.179} C_VEL
LIN {X 0,Y 446.405,Z 282.501,A -85,B 0,C 180,E1 -8851.301,E2 -8851.301} C_VEL
LIN {X 0,Y 446.414,Z 282.502,A -85,B 0,C 180,E1 -8854.524,E2 -8854.524} C_VEL
LIN {X 0,Y 446.407,Z 282.498,A -85,B 0,C 180,E1 -8858.08,E2 -8858.08} C_VEL
LIN {X 0,Y 446.42,Z 282.504,A -85,B 0,C 180,E1 -8860.918,E2 -8860.918} C_VEL
LIN {X 0,Y 446.392,Z 282.503,A -85,B 0,C 180,E1 -8863.847,E2 -8863.847} C_VEL
LIN {X 0,Y 446.393,Z 282.507,A -85,B 0,C 180,E1 -8866.404,E2 -8866.404} C_VEL
LIN {X 0,Y 446.423,Z 282.504,A -85,B 0,C 180,E1 -8869.083,E2 -8869.083} C_VEL
LIN {X 0,Y 446.411,Z 282.498,A -85,B 0,C 180,E1 -8871.922,E2 -8871.922} C_VEL
LIN {X 0,Y 446.42,Z 282.501,A -85,B 0,C 180,E1 -8875.477,E2 -8875.477} C_VEL
LIN {X 0,Y 446.413,Z 282.502,A -85,B 0,C 180,E1 -8878.7,E2 -8878.7} C_VEL
LIN {X 0,Y 446.5,Z 282.515,A -85,B 0,C 180,E1 -8881.954,E2 -8881.954} C_VEL
LIN {X 0,Y 449.584,Z 295.886,A -85,B 0,C 180,E1 -8884.644,E2 -8884.644} C_VEL
LIN {X 0,Y 449.848,Z 296.817,A -85,B 0,C 180,E1 -8884.718,E2 -8884.718} C_VEL
LIN {X 0,Y 453.69,Z 306.582,A -85,B 0,C 180,E1 -8885.116,E2 -8885.116} C_VEL
LIN {X 0,Y 456.626,Z 319.641,A -85,B 0,C 180,E1 -8885.51,E2 -8885.51} C_VEL
LIN {X 0,Y 455.105,Z 428.391,A -85,B 0,C 180,E1 -8887.261,E2 -8887.261} C_VEL
LIN {X 0,Y 454.88,Z 446.918,A -85,B 0,C 180,E1 -8887.56,E2 -8887.56} C_VEL
LIN {X 0,Y 454.187,Z 452.764,A -85,B 0,C 180,E1 -8887.621,E2 -8887.621} C_VEL
LIN {X 0,Y 448.871,Z 469.779,A -85,B 0,C 180,E1 -8887.736,E2 -8887.736} C_VEL
LIN {X 0,Y 447.68,Z 475.473,A -85,B 0,C 180,E1 -8887.862,E2 -8887.862} C_VEL
LIN {X 0,Y 447.511,Z 477.373,A -85,B 0,C 180,E1 -8887.923,E2 -8887.923} C_VEL
LIN {X 0,Y 447,Z 490.135,A -85,B 0,C 180,E1 -8888.446,E2 -8888.446} C_VEL
LIN {X 0,Y 446.143,Z 503.147,A -85,B 0,C 180,E1 -8889.121,E2 -8889.121} C_VEL
LIN {X 0,Y 445.182,Z 517.133,A -85,B 0,C 180,E1 -8890.039,E2 -8890.039} C_VEL
LIN {X 0,Y 444.133,Z 529.913,A -85,B 0,C 180,E1 -8891.072,E2 -8891.072} C_VEL
LIN {X 0,Y 443.136,Z 542.032,A -85,B 0,C 180,E1 -8892.26,E2 -8892.26} C_VEL
LIN {X 0,Y 442.077,Z 553.533,A -85,B 0,C 180,E1 -8893.61,E2 -8893.61} C_VEL
LIN {X 0,Y 441.221,Z 563.469,A -85,B 0,C 180,E1 -8894.999,E2 -8894.999} C_VEL
LIN {X 0,Y 440.429,Z 572.038,A -85,B 0,C 180,E1 -8896.411,E2 -8896.411} C_VEL
LIN {X 0,Y 439.811,Z 580.163,A -85,B 0,C 180,E1 -8898.011,E2 -8898.011} C_VEL
LIN {X 0,Y 439.183,Z 587.921,A -85,B 0,C 180,E1 -8899.862,E2 -8899.862} C_VEL
LIN {X 0,Y 438.813,Z 594.095,A -85,B 0,C 180,E1 -8901.713,E2 -8901.713} C_VEL
LIN {X 0,Y 438.593,Z 598.862,A -85,B 0,C 180,E1 -8903.56,E2 -8903.56} C_VEL
LIN {X 0,Y 438.361,Z 602.358,A -85,B 0,C 180,E1 -8905.402,E2 -8905.402} C_VEL
LIN {X 0,Y 438.381,Z 604.667,A -85,B 0,C 180,E1 -8907.243,E2 -8907.243} C_VEL
LIN {X 0,Y 438.252,Z 605.851,A -85,B 0,C 180,E1 -8909.081,E2 -8909.081} C_VEL
LIN {X 0,Y 438.253,Z 605.868,A -85,B 0,C 180,E1 -8910.919,E2 -8910.919} C_VEL
LIN {X 0,Y 438.379,Z 604.75,A -85,B 0,C 180,E1 -8912.757,E2 -8912.757} C_VEL
LIN {X 0,Y 438.359,Z 602.507,A -85,B 0,C 180,E1 -8914.598,E2 -8914.598} C_VEL
LIN {X 0,Y 438.545,Z 598.967,A -85,B 0,C 180,E1 -8916.488,E2 -8916.488} C_VEL
LIN {X 0,Y 438.812,Z 594.373,A -85,B 0,C 180,E1 -8918.287,E2 -8918.287} C_VEL
LIN {X 0,Y 439.161,Z 588.283,A -85,B 0,C 180,E1 -8920.139,E2 -8920.139} C_VEL
LIN {X 0,Y 439.78,Z 580.609,A -85,B 0,C 180,E1 -8921.99,E2 -8921.99} C_VEL
LIN {X 0,Y 440.409,Z 572.555,A -85,B 0,C 180,E1 -8923.59,E2 -8923.59} C_VEL
LIN {X 0,Y 441.283,Z 562.569,A -85,B 0,C 180,E1 -8925.235,E2 -8925.235} C_VEL
LIN {X 0,Y 442.168,Z 552.458,A -85,B 0,C 180,E1 -8926.624,E2 -8926.624} C_VEL
LIN {X 0,Y 443.14,Z 541.403,A -85,B 0,C 180,E1 -8927.904,E2 -8927.904} C_VEL
LIN {X 0,Y 444.144,Z 529.628,A -85,B 0,C 180,E1 -8929.048,E2 -8929.048} C_VEL
LIN {X 0,Y 445.239,Z 516.792,A -85,B 0,C 180,E1 -8930.079,E2 -8930.079} C_VEL
LIN {X 0,Y 446.199,Z 502.714,A -85,B 0,C 180,E1 -8930.997,E2 -8930.997} C_VEL
LIN {X 0,Y 447.065,Z 487.757,A -85,B 0,C 180,E1 -8931.755,E2 -8931.755} C_VEL
LIN {X 0,Y 447.69,Z 472.887,A -85,B 0,C 180,E1 -8932.315,E2 -8932.315} C_VEL
LIN {X 0,Y 448.147,Z 458.313,A -85,B 0,C 180,E1 -8932.686,E2 -8932.686} C_VEL
LIN {X 0,Y 449.288,Z 382.332,A -85,B 0,C 180,E1 -8933.936,E2 -8933.936} C_VEL
LIN {X 0,Y 450.068,Z 319.959,A -85,B 0,C 180,E1 -8934.964,E2 -8934.964} C_VEL
LIN {X 0,Y 447.088,Z 307.426,A -85,B 0,C 180,E1 -8935.362,E2 -8935.362} C_VEL
LIN {X 0,Y 442.461,Z 296.241,A -85,B 0,C 180,E1 -8935.863,E2 -8935.863} C_VEL
LIN {X 0,Y 439.925,Z 285.459,A -85,B 0,C 180,E1 -8938.071,E2 -8938.071} C_VEL
LIN {X 0,Y 439.425,Z 283.375,A -85,B 0,C 180,E1 -8938.537,E2 -8938.537} C_VEL
LIN {X 0,Y 439.368,Z 283.381,A -85,B 0,C 180,E1 -8942.03,E2 -8942.03} C_VEL
LIN {X 0,Y 439.393,Z 283.382,A -85,B 0,C 180,E1 -8945.34,E2 -8945.34} C_VEL
LIN {X 0,Y 439.378,Z 283.381,A -85,B 0,C 180,E1 -8948.594,E2 -8948.594} C_VEL
LIN {X 0,Y 439.384,Z 283.377,A -85,B 0,C 180,E1 -8951.256,E2 -8951.256} C_VEL
LIN {X 0,Y 439.394,Z 283.377,A -85,B 0,C 180,E1 -8954.729,E2 -8954.729} C_VEL
LIN {X 0,Y 439.378,Z 283.367,A -85,B 0,C 180,E1 -8957.793,E2 -8957.793} C_VEL
LIN {X 0,Y 439.382,Z 283.376,A -85,B 0,C 180,E1 -8960.222,E2 -8960.222} C_VEL
LIN {X 0,Y 439.365,Z 283.371,A -85,B 0,C 180,E1 -8963.712,E2 -8963.712} C_VEL
LIN {X 0,Y 439.362,Z 283.381,A -85,B 0,C 180,E1 -8967.053,E2 -8967.053} C_VEL
LIN {X 0,Y 439.371,Z 283.367,A -85,B 0,C 180,E1 -8970.273,E2 -8970.273} C_VEL
LIN {X 0,Y 439.409,Z 283.373,A -85,B 0,C 180,E1 -8973.395,E2 -8973.395} C_VEL
LIN {X 0,Y 439.371,Z 283.378,A -85,B 0,C 180,E1 -8976.429,E2 -8976.429} C_VEL
LIN {X 0,Y 439.377,Z 283.379,A -85,B 0,C 180,E1 -8979.396,E2 -8979.396} C_VEL
LIN {X 0,Y 439.393,Z 283.372,A -85,B 0,C 180,E1 -8982.308,E2 -8982.308} C_VEL
LIN {X 0,Y 439.433,Z 283.37,A -85,B 0,C 180,E1 -8985.173,E2 -8985.173} C_VEL
LIN {X 0,Y 439.47,Z 283.363,A -85,B 0,C 180,E1 -8988.001,E2 -8988.001} C_VEL
LIN {X 0,Y 439.491,Z 283.359,A -85,B 0,C 180,E1 -8991.725,E2 -8991.725} C_VEL
LIN {X 0,Y 439.595,Z 283.353,A -85,B 0,C 180,E1 -8994.495,E2 -8994.495} C_VEL
LIN {X 0,Y 439.62,Z 283.348,A -85,B 0,C 180,E1 -8998.168,E2 -8998.168} C_VEL
LIN {X 0,Y 439.743,Z 283.327,A -85,B 0,C 180,E1 -9000,E2 -9000} C_VEL
LIN {X 0,Y 439.598,Z 283.353,A -85,B 0,C 180,E1 -9002.749,E2 -9002.749} C_VEL
LIN {X 0,Y 439.583,Z 283.354,A -85,B 0,C 180,E1 -9006.426,E2 -9006.426} C_VEL
LIN {X 0,Y 439.471,Z 283.361,A -85,B 0,C 180,E1 -9009.202,E2 -9009.202} C_VEL
LIN {X 0,Y 439.454,Z 283.364,A -85,B 0,C 180,E1 -9012.938,E2 -9012.938} C_VEL
LIN {X 0,Y 439.433,Z 283.376,A -85,B 0,C 180,E1 -9016.347,E2 -9016.347} C_VEL
LIN {X 0,Y 439.39,Z 283.376,A -85,B 0,C 180,E1 -9019.627,E2 -9019.627} C_VEL
LIN {X 0,Y 439.35,Z 283.383,A -85,B 0,C 180,E1 -9022.576,E2 -9022.576} C_VEL
LIN {X 0,Y 439.351,Z 283.379,A -85,B 0,C 180,E1 -9025.588,E2 -9025.588} C_VEL
LIN {X 0,Y 439.387,Z 283.378,A -85,B 0,C 180,E1 -9028.676,E2 -9028.676} C_VEL
LIN {X 0,Y 439.356,Z 283.385,A -85,B 0,C 180,E1 -9032.03,E2 -9032.03} C_VEL
LIN {X 0,Y 439.376,Z 283.377,A -85,B 0,C 180,E1 -9035.339,E2 -9035.339} C_VEL
LIN {X 0,Y 439.345,Z 283.38,A -85,B 0,C 180,E1 -9038.599,E2 -9038.599} C_VEL
LIN {X 0,Y 439.35,Z 283.381,A -85,B 0,C 180,E1 -9042.21,E2 -9042.21} C_VEL
LIN {X 0,Y 439.368,Z 283.379,A -85,B 0,C 180,E1 -9045.268,E2 -9045.268} C_VEL
LIN {X 0,Y 439.356,Z 283.38,A -85,B 0,C 180,E1 -9048.748,E2 -9048.748} C_VEL
LIN {X 0,Y 439.351,Z 283.382,A -85,B 0,C 180,E1 -9051.612,E2 -9051.612} C_VEL
LIN {X 0,Y 439.392,Z 283.377,A -85,B 0,C 180,E1 -9054.845,E2 -9054.845} C_VEL
LIN {X 0,Y 439.404,Z 283.534,A -85,B 0,C 180,E1 -9058.177,E2 -9058.177} C_VEL
LIN {X 0,Y 442.905,Z 297.474,A -85,B 0,C 180,E1 -9060.778,E2 -9060.778} C_VEL
LIN {X 0,Y 444.965,Z 306.806,A -85,B 0,C 180,E1 -9062.444,E2 -9062.444} C_VEL
LIN {X 0,Y 444.159,Z 318.478,A -85,B 0,C 180,E1 -9064.288,E2 -9064.288} C_VEL
LIN {X 0,Y 449.782,Z 346.941,A -85,B 0,C 180,E1 -9065.127,E2 -9065.127} C_VEL
LIN {X 0,Y 448.477,Z 449.731,A -85,B 0,C 180,E1 -9066.814,E2 -9066.814} C_VEL
LIN {X 0,Y 447.81,Z 485.553,A -85,B 0,C 180,E1 -9067.418,E2 -9067.418} C_VEL
LIN {X 0,Y 447.221,Z 501.13,A -85,B 0,C 180,E1 -9067.862,E2 -9067.862} C_VEL
LIN {X 0,Y 446.415,Z 515.526,A -85,B 0,C 180,E1 -9068.445,E2 -9068.445} C_VEL
LIN {X 0,Y 445.53,Z 529.768,A -85,B 0,C 180,E1 -9069.212,E2 -9069.212} C_VEL
LIN {X 0,Y 444.466,Z 543.271,A -85,B 0,C 180,E1 -9070.126,E2 -9070.126} C_VEL
LIN {X 0,Y 443.286,Z 557.022,A -85,B 0,C 180,E1 -9071.274,E2 -9071.274} C_VEL
LIN {X 0,Y 442.256,Z 568.639,A -85,B 0,C 180,E1 -9072.453,E2 -9072.453} C_VEL
LIN {X 0,Y 441.295,Z 579.917,A -85,B 0,C 180,E1 -9073.818,E2 -9073.818} C_VEL
LIN {X 0,Y 440.493,Z 589.615,A -85,B 0,C 180,E1 -9075.21,E2 -9075.21} C_VEL
LIN {X 0,Y 439.689,Z 599.141,A -85,B 0,C 180,E1 -9076.834,E2 -9076.834} C_VEL
LIN {X 0,Y 439.245,Z 607.085,A -85,B 0,C 180,E1 -9078.463,E2 -9078.463} C_VEL
LIN {X 0,Y 438.713,Z 614.498,A -85,B 0,C 180,E1 -9080.317,E2 -9080.317} C_VEL
LIN {X 0,Y 438.487,Z 620.384,A -85,B 0,C 180,E1 -9082.17,E2 -9082.17} C_VEL
LIN {X 0,Y 438.363,Z 624.272,A -85,B 0,C 180,E1 -9083.724,E2 -9083.724} C_VEL
LIN {X 0,Y 438.292,Z 627.42,A -85,B 0,C 180,E1 -9085.402,E2 -9085.402} C_VEL
LIN {X 0,Y 438.326,Z 629.748,A -85,B 0,C 180,E1 -9087.243,E2 -9087.243} C_VEL
LIN {X 0,Y 438.249,Z 630.917,A -85,B 0,C 180,E1 -9089.081,E2 -9089.081} C_VEL
LIN {X 0,Y 438.249,Z 630.916,A -85,B 0,C 180,E1 -9090.919,E2 -9090.919} C_VEL
LIN {X 0,Y 438.326,Z 629.742,A -85,B 0,C 180,E1 -9092.757,E2 -9092.757} C_VEL
LIN {X 0,Y 438.291,Z 627.412,A -85,B 0,C 180,E1 -9094.598,E2 -9094.598} C_VEL
LIN {X 0,Y 438.357,Z 623.879,A -85,B 0,C 180,E1 -9096.444,E2 -9096.444} C_VEL
LIN {X 0,Y 438.549,Z 619.055,A -85,B 0,C 180,E1 -9098.292,E2 -9098.292} C_VEL
LIN {X 0,Y 438.787,Z 612.805,A -85,B 0,C 180,E1 -9100.147,E2 -9100.147} C_VEL
LIN {X 0,Y 439.252,Z 606.051,A -85,B 0,C 180,E1 -9101.771,E2 -9101.771} C_VEL
LIN {X 0,Y 439.843,Z 597.887,A -85,B 0,C 180,E1 -9103.396,E2 -9103.396} C_VEL
LIN {X 0,Y 440.617,Z 588.103,A -85,B 0,C 180,E1 -9105.022,E2 -9105.022} C_VEL
LIN {X 0,Y 441.518,Z 578.104,A -85,B 0,C 180,E1 -9106.411,E2 -9106.411} C_VEL
LIN {X 0,Y 442.524,Z 566.447,A -85,B 0,C 180,E1 -9107.777,E2 -9107.777} C_VEL
LIN {X 0,Y 443.499,Z 554.401,A -85,B 0,C 180,E1 -9108.956,E2 -9108.956} C_VEL
LIN {X 0,Y 444.58,Z 541.632,A -85,B 0,C 180,E1 -9109.989,E2 -9109.989} C_VEL
LIN {X 0,Y 445.633,Z 527.706,A -85,B 0,C 180,E1 -9110.904,E2 -9110.904} C_VEL
LIN {X 0,Y 446.554,Z 513.389,A -85,B 0,C 180,E1 -9111.645,E2 -9111.645} C_VEL
LIN {X 0,Y 447.251,Z 498.767,A -85,B 0,C 180,E1 -9112.216,E2 -9112.216} C_VEL
LIN {X 0,Y 447.868,Z 484.042,A -85,B 0,C 180,E1 -9112.609,E2 -9112.609} C_VEL
LIN {X 0,Y 449.903,Z 348.198,A -85,B 0,C 180,E1 -9114.839,E2 -9114.839} C_VEL
LIN {X 0,Y 444.198,Z 318.456,A -85,B 0,C 180,E1 -9115.707,E2 -9115.707} C_VEL
LIN {X 0,Y 444.956,Z 306.785,A -85,B 0,C 180,E1 -9117.553,E2 -9117.553} C_VEL
LIN {X 0,Y 442.573,Z 295.961,A -85,B 0,C 180,E1 -9119.489,E2 -9119.489} C_VEL
LIN {X 0,Y 439.368,Z 283.373,A -85,B 0,C 180,E1 -9121.86,E2 -9121.86} C_VEL
LIN {X 0,Y 439.392,Z 283.376,A -85,B 0,C 180,E1 -9125.155,E2 -9125.155} C_VEL
LIN {X 0,Y 439.349,Z 283.385,A -85,B 0,C 180,E1 -9128.597,E2 -9128.597} C_VEL
LIN {X 0,Y 439.344,Z 283.387,A -85,B 0,C 180,E1 -9132.209,E2 -9132.209} C_VEL
LIN {X 0,Y 439.368,Z 283.379,A -85,B 0,C 180,E1 -9135.267,E2 -9135.267} C_VEL
LIN {X 0,Y 439.359,Z 283.379,A -85,B 0,C 180,E1 -9138.746,E2 -9138.746} C_VEL
LIN {X 0,Y 439.347,Z 283.384,A -85,B 0,C 180,E1 -9141.61,E2 -9141.61} C_VEL
LIN {X 0,Y 439.381,Z 283.374,A -85,B 0,C 180,E1 -9144.842,E2 -9144.842} C_VEL
LIN {X 0,Y 439.359,Z 283.382,A -85,B 0,C 180,E1 -9148.139,E2 -9148.139} C_VEL
LIN {X 0,Y 439.391,Z 283.379,A -85,B 0,C 180,E1 -9151.605,E2 -9151.605} C_VEL
LIN {X 0,Y 439.351,Z 283.38,A -85,B 0,C 180,E1 -9154.412,E2 -9154.412} C_VEL
LIN {X 0,Y 439.351,Z 283.383,A -85,B 0,C 180,E1 -9157.424,E2 -9157.424} C_VEL
LIN {X 0,Y 439.429,Z 283.356,A -85,B 0,C 180,E1 -9160.663,E2 -9160.663} C_VEL
LIN {X 0,Y 439.448,Z 283.368,A -85,B 0,C 180,E1 -9164.224,E2 -9164.224} C_VEL
LIN {X 0,Y 439.462,Z 283.347,A -85,B 0,C 180,E1 -9168.001,E2 -9168.001} C_VEL
LIN {X 0,Y 439.466,Z 283.37,A -85,B 0,C 180,E1 -9171.725,E2 -9171.725} C_VEL
LIN {X 0,Y 439.594,Z 283.344,A -85,B 0,C 180,E1 -9174.496,E2 -9174.496} C_VEL
LIN {X 0,Y 439.612,Z 283.342,A -85,B 0,C 180,E1 -9178.168,E2 -9178.168} C_VEL
LIN {X 0,Y 439.636,Z 283.345,A -85,B 0,C 180,E1 -9180,E2 -9180} C_VEL
LIN {X 0,Y 439.603,Z 283.345,A -85,B 0,C 180,E1 -9182.749,E2 -9182.749} C_VEL
LIN {X 0,Y 439.585,Z 283.347,A -85,B 0,C 180,E1 -9186.426,E2 -9186.426} C_VEL
LIN {X 0,Y 439.481,Z 283.37,A -85,B 0,C 180,E1 -9189.202,E2 -9189.202} C_VEL
LIN {X 0,Y 439.453,Z 283.37,A -85,B 0,C 180,E1 -9192.938,E2 -9192.938} C_VEL
LIN {X 0,Y 439.435,Z 283.369,A -85,B 0,C 180,E1 -9196.348,E2 -9196.348} C_VEL
LIN {X 0,Y 439.391,Z 283.362,A -85,B 0,C 180,E1 -9199.627,E2 -9199.627} C_VEL
LIN {X 0,Y 439.352,Z 283.375,A -85,B 0,C 180,E1 -9202.576,E2 -9202.576} C_VEL
LIN {X 0,Y 439.376,Z 283.373,A -85,B 0,C 180,E1 -9205.587,E2 -9205.587} C_VEL
LIN {X 0,Y 439.408,Z 283.366,A -85,B 0,C 180,E1 -9208.674,E2 -9208.674} C_VEL
LIN {X 0,Y 439.356,Z 283.376,A -85,B 0,C 180,E1 -9212.03,E2 -9212.03} C_VEL
LIN {X 0,Y 439.384,Z 283.377,A -85,B 0,C 180,E1 -9215.341,E2 -9215.341} C_VEL
LIN {X 0,Y 439.37,Z 283.379,A -85,B 0,C 180,E1 -9218.597,E2 -9218.597} C_VEL
LIN {X 0,Y 439.382,Z 283.378,A -85,B 0,C 180,E1 -9221.258,E2 -9221.258} C_VEL
LIN {X 0,Y 439.393,Z 283.378,A -85,B 0,C 180,E1 -9224.73,E2 -9224.73} C_VEL
LIN {X 0,Y 439.391,Z 283.376,A -85,B 0,C 180,E1 -9227.797,E2 -9227.797} C_VEL
LIN {X 0,Y 439.432,Z 283.373,A -85,B 0,C 180,E1 -9230.229,E2 -9230.229} C_VEL
LIN {X 0,Y 439.369,Z 283.377,A -85,B 0,C 180,E1 -9233.714,E2 -9233.714} C_VEL
LIN {X 0,Y 439.369,Z 283.379,A -85,B 0,C 180,E1 -9237.055,E2 -9237.055} C_VEL
LIN {X 0,Y 439.38,Z 283.381,A -85,B 0,C 180,E1 -9240.275,E2 -9240.275} C_VEL
LIN {X 0,Y 439.431,Z 283.429,A -85,B 0,C 180,E1 -9241.599,E2 -9241.599} C_VEL
LIN {X 0,Y 442.242,Z 295.206,A -85,B 0,C 180,E1 -9244.025,E2 -9244.025} C_VEL
LIN {X 0,Y 442.571,Z 296.67,A -85,B 0,C 180,E1 -9244.265,E2 -9244.265} C_VEL
LIN {X 0,Y 447.653,Z 309.375,A -85,B 0,C 180,E1 -9244.802,E2 -9244.802} C_VEL
LIN {X 0,Y 450.2,Z 321.321,A -85,B 0,C 180,E1 -9245.162,E2 -9245.162} C_VEL
LIN {X 0,Y 448.454,Z 437.553,A -85,B 0,C 180,E1 -9247.057,E2 -9247.057} C_VEL
LIN {X 0,Y 448.024,Z 462.34,A -85,B 0,C 180,E1 -9247.49,E2 -9247.49} C_VEL
LIN {X 0,Y 447.511,Z 477.373,A -85,B 0,C 180,E1 -9247.923,E2 -9247.923} C_VEL
LIN {X 0,Y 446.567,Z 483.051,A -85,B 0,C 180,E1 -9248.099,E2 -9248.099} C_VEL
LIN {X 0,Y 443.37,Z 492.245,A -85,B 0,C 180,E1 -9248.358,E2 -9248.358} C_VEL
LIN {X 0,Y 440.241,Z 501.301,A -85,B 0,C 180,E1 -9248.698,E2 -9248.698} C_VEL
LIN {X 0,Y 439.291,Z 506.644,A -85,B 0,C 180,E1 -9248.987,E2 -9248.987} C_VEL
LIN {X 0,Y 438.26,Z 520.479,A -85,B 0,C 180,E1 -9249.955,E2 -9249.955} C_VEL
LIN {X 0,Y 437.066,Z 533.947,A -85,B 0,C 180,E1 -9251.119,E2 -9251.119} C_VEL
LIN {X 0,Y 436.01,Z 546.157,A -85,B 0,C 180,E1 -9252.409,E2 -9252.409} C_VEL
LIN {X 0,Y 434.926,Z 557.278,A -85,B 0,C 180,E1 -9253.815,E2 -9253.815} C_VEL
LIN {X 0,Y 433.884,Z 568.079,A -85,B 0,C 180,E1 -9255.46,E2 -9255.46} C_VEL
LIN {X 0,Y 433.034,Z 576.601,A -85,B 0,C 180,E1 -9257.019,E2 -9257.019} C_VEL
LIN {X 0,Y 432.582,Z 583.459,A -85,B 0,C 180,E1 -9258.521,E2 -9258.521} C_VEL
LIN {X 0,Y 432.044,Z 589.8,A -85,B 0,C 180,E1 -9260.166,E2 -9260.166} C_VEL
LIN {X 0,Y 431.693,Z 595.621,A -85,B 0,C 180,E1 -9262.046,E2 -9262.046} C_VEL
LIN {X 0,Y 431.522,Z 599.066,A -85,B 0,C 180,E1 -9263.454,E2 -9263.454} C_VEL
LIN {X 0,Y 431.29,Z 602.561,A -85,B 0,C 180,E1 -9265.327,E2 -9265.327} C_VEL
LIN {X 0,Y 431.31,Z 604.87,A -85,B 0,C 180,E1 -9267.198,E2 -9267.198} C_VEL
LIN {X 0,Y 431.169,Z 606.054,A -85,B 0,C 180,E1 -9269.066,E2 -9269.066} C_VEL
LIN {X 0,Y 431.17,Z 606.07,A -85,B 0,C 180,E1 -9270.934,E2 -9270.934} C_VEL
LIN {X 0,Y 431.307,Z 604.952,A -85,B 0,C 180,E1 -9272.802,E2 -9272.802} C_VEL
LIN {X 0,Y 431.288,Z 602.709,A -85,B 0,C 180,E1 -9274.673,E2 -9274.673} C_VEL
LIN {X 0,Y 431.481,Z 599.275,A -85,B 0,C 180,E1 -9276.547,E2 -9276.547} C_VEL
LIN {X 0,Y 431.755,Z 594.575,A -85,B 0,C 180,E1 -9278.424,E2 -9278.424} C_VEL
LIN {X 0,Y 432.124,Z 588.485,A -85,B 0,C 180,E1 -9280.306,E2 -9280.306} C_VEL
LIN {X 0,Y 432.803,Z 580.811,A -85,B 0,C 180,E1 -9282.186,E2 -9282.186} C_VEL
LIN {X 0,Y 433.446,Z 572.757,A -85,B 0,C 180,E1 -9283.813,E2 -9283.813} C_VEL
LIN {X 0,Y 434.388,Z 562.771,A -85,B 0,C 180,E1 -9285.483,E2 -9285.483} C_VEL
LIN {X 0,Y 435.332,Z 552.659,A -85,B 0,C 180,E1 -9286.893,E2 -9286.893} C_VEL
LIN {X 0,Y 436.469,Z 540.647,A -85,B 0,C 180,E1 -9288.296,E2 -9288.296} C_VEL
LIN {X 0,Y 437.582,Z 528.54,A -85,B 0,C 180,E1 -9289.467,E2 -9289.467} C_VEL
LIN {X 0,Y 438.668,Z 515.415,A -85,B 0,C 180,E1 -9290.515,E2 -9290.515} C_VEL
LIN {X 0,Y 439.583,Z 502.91,A -85,B 0,C 180,E1 -9291.328,E2 -9291.328} C_VEL
LIN {X 0,Y 440.451,Z 488.665,A -85,B 0,C 180,E1 -9292.065,E2 -9292.065} C_VEL
LIN {X 0,Y 441.104,Z 473.99,A -85,B 0,C 180,E1 -9292.635,E2 -9292.635} C_VEL
LIN {X 0,Y 441.57,Z 459.996,A -85,B 0,C 180,E1 -9293.012,E2 -9293.012} C_VEL
LIN {X 0,Y 442.817,Z 382.508,A -85,B 0,C 180,E1 -9294.308,E2 -9294.308} C_VEL
LIN {X 0,Y 443.648,Z 321.236,A -85,B 0,C 180,E1 -9295.331,E2 -9295.331} C_VEL
LIN {X 0,Y 440.883,Z 309.817,A -85,B 0,C 180,E1 -9295.705,E2 -9295.705} C_VEL
LIN {X 0,Y 435.285,Z 296.485,A -85,B 0,C 180,E1 -9296.317,E2 -9296.317} C_VEL
LIN {X 0,Y 432.361,Z 284.256,A -85,B 0,C 180,E1 -9298.903,E2 -9298.903} C_VEL
LIN {X 0,Y 432.323,Z 284.259,A -85,B 0,C 180,E1 -9302.292,E2 -9302.292} C_VEL
LIN {X 0,Y 432.338,Z 284.256,A -85,B 0,C 180,E1 -9304.676,E2 -9304.676} C_VEL
LIN {X 0,Y 432.34,Z 284.258,A -85,B 0,C 180,E1 -9308.148,E2 -9308.148} C_VEL
LIN {X 0,Y 432.328,Z 284.261,A -85,B 0,C 180,E1 -9311.601,E2 -9311.601} C_VEL
LIN {X 0,Y 432.328,Z 284.255,A -85,B 0,C 180,E1 -9314.346,E2 -9314.346} C_VEL
LIN {X 0,Y 432.311,Z 284.258,A -85,B 0,C 180,E1 -9317.015,E2 -9317.015} C_VEL
LIN {X 0,Y 432.325,Z 284.256,A -85,B 0,C 180,E1 -9319.82,E2 -9319.82} C_VEL
LIN {X 0,Y 432.298,Z 284.25,A -85,B 0,C 180,E1 -9323.021,E2 -9323.021} C_VEL
LIN {X 0,Y 432.325,Z 284.255,A -85,B 0,C 180,E1 -9326.001,E2 -9326.001} C_VEL
LIN {X 0,Y 432.336,Z 284.242,A -85,B 0,C 180,E1 -9329.49,E2 -9329.49} C_VEL
LIN {X 0,Y 432.376,Z 284.254,A -85,B 0,C 180,E1 -9332.927,E2 -9332.927} C_VEL
LIN {X 0,Y 432.355,Z 284.251,A -85,B 0,C 180,E1 -9336.022,E2 -9336.022} C_VEL
LIN {X 0,Y 432.339,Z 284.255,A -85,B 0,C 180,E1 -9339.045,E2 -9339.045} C_VEL
LIN {X 0,Y 432.348,Z 284.248,A -85,B 0,C 180,E1 -9342.01,E2 -9342.01} C_VEL
LIN {X 0,Y 432.382,Z 284.252,A -85,B 0,C 180,E1 -9344.926,E2 -9344.926} C_VEL
LIN {X 0,Y 432.447,Z 284.238,A -85,B 0,C 180,E1 -9347.803,E2 -9347.803} C_VEL
LIN {X 0,Y 432.451,Z 284.236,A -85,B 0,C 180,E1 -9351.589,E2 -9351.589} C_VEL
LIN {X 0,Y 432.572,Z 284.227,A -85,B 0,C 180,E1 -9354.406,E2 -9354.406} C_VEL
LIN {X 0,Y 432.59,Z 284.223,A -85,B 0,C 180,E1 -9358.138,E2 -9358.138} C_VEL
LIN {X 0,Y 432.713,Z 284.203,A -85,B 0,C 180,E1 -9360,E2 -9360} C_VEL
LIN {X 0,Y 432.551,Z 284.23,A -85,B 0,C 180,E1 -9362.794,E2 -9362.794} C_VEL
LIN {X 0,Y 432.571,Z 284.222,A -85,B 0,C 180,E1 -9365.594,E2 -9365.594} C_VEL
LIN {X 0,Y 432.448,Z 284.242,A -85,B 0,C 180,E1 -9368.41,E2 -9368.41} C_VEL
LIN {X 0,Y 432.446,Z 284.245,A -85,B 0,C 180,E1 -9372.197,E2 -9372.197} C_VEL
LIN {X 0,Y 432.414,Z 284.248,A -85,B 0,C 180,E1 -9376.039,E2 -9376.039} C_VEL
LIN {X 0,Y 432.375,Z 284.25,A -85,B 0,C 180,E1 -9379.485,E2 -9379.485} C_VEL
LIN {X 0,Y 432.298,Z 284.26,A -85,B 0,C 180,E1 -9382.965,E2 -9382.965} C_VEL
LIN {X 0,Y 432.305,Z 284.258,A -85,B 0,C 180,E1 -9386.036,E2 -9386.036} C_VEL
LIN {X 0,Y 432.322,Z 284.256,A -85,B 0,C 180,E1 -9389.189,E2 -9389.189} C_VEL
LIN {X 0,Y 432.312,Z 284.256,A -85,B 0,C 180,E1 -9392.444,E2 -9392.444} C_VEL
LIN {X 0,Y 432.323,Z 284.259,A -85,B 0,C 180,E1 -9395.819,E2 -9395.819} C_VEL
LIN {X 0,Y 432.291,Z 284.257,A -85,B 0,C 180,E1 -9399.349,E2 -9399.349} C_VEL
LIN {X 0,Y 432.301,Z 284.252,A -85,B 0,C 180,E1 -9401.801,E2 -9401.801} C_VEL
LIN {X 0,Y 432.325,Z 284.258,A -85,B 0,C 180,E1 -9404.348,E2 -9404.348} C_VEL
LIN {X 0,Y 432.295,Z 284.259,A -85,B 0,C 180,E1 -9407.019,E2 -9407.019} C_VEL
LIN {X 0,Y 432.282,Z 284.263,A -85,B 0,C 180,E1 -9409.829,E2 -9409.829} C_VEL
LIN {X 0,Y 432.293,Z 284.259,A -85,B 0,C 180,E1 -9413.022,E2 -9413.022} C_VEL
LIN {X 0,Y 432.355,Z 284.257,A -85,B 0,C 180,E1 -9415.997,E2 -9415.997} C_VEL
LIN {X 0,Y 432.317,Z 284.305,A -85,B 0,C 180,E1 -9417.763,E2 -9417.763} C_VEL
LIN {X 0,Y 435.79,Z 297.848,A -85,B 0,C 180,E1 -9420.352,E2 -9420.352} C_VEL
LIN {X 0,Y 438.112,Z 308.418,A -85,B 0,C 180,E1 -9422.277,E2 -9422.277} C_VEL
LIN {X 0,Y 437.478,Z 318.55,A -85,B 0,C 180,E1 -9423.877,E2 -9423.877} C_VEL
LIN {X 0,Y 443.345,Z 348.103,A -85,B 0,C 180,E1 -9424.764,E2 -9424.764} C_VEL
LIN {X 0,Y 441.915,Z 451.336,A -85,B 0,C 180,E1 -9426.48,E2 -9426.48} C_VEL
LIN {X 0,Y 441.254,Z 485.361,A -85,B 0,C 180,E1 -9427.063,E2 -9427.063} C_VEL
LIN {X 0,Y 440.629,Z 500.973,A -85,B 0,C 180,E1 -9427.514,E2 -9427.514} C_VEL
LIN {X 0,Y 439.756,Z 515.968,A -85,B 0,C 180,E1 -9428.136,E2 -9428.136} C_VEL
LIN {X 0,Y 438.866,Z 529.569,A -85,B 0,C 180,E1 -9428.881,E2 -9428.881} C_VEL
LIN {X 0,Y 437.74,Z 543.07,A -85,B 0,C 180,E1 -9429.807,E2 -9429.807} C_VEL
LIN {X 0,Y 436.512,Z 556.82,A -85,B 0,C 180,E1 -9430.972,E2 -9430.972} C_VEL
LIN {X 0,Y 435.376,Z 569.176,A -85,B 0,C 180,E1 -9432.25,E2 -9432.25} C_VEL
LIN {X 0,Y 434.234,Z 581.484,A -85,B 0,C 180,E1 -9433.789,E2 -9433.789} C_VEL
LIN {X 0,Y 433.312,Z 592.349,A -85,B 0,C 180,E1 -9435.44,E2 -9435.44} C_VEL
LIN {X 0,Y 432.433,Z 601.907,A -85,B 0,C 180,E1 -9437.195,E2 -9437.195} C_VEL
LIN {X 0,Y 432.101,Z 608.913,A -85,B 0,C 180,E1 -9438.745,E2 -9438.745} C_VEL
LIN {X 0,Y 431.589,Z 615.92,A -85,B 0,C 180,E1 -9440.628,E2 -9440.628} C_VEL
LIN {X 0,Y 431.385,Z 621.435,A -85,B 0,C 180,E1 -9442.511,E2 -9442.511} C_VEL
LIN {X 0,Y 431.222,Z 625.603,A -85,B 0,C 180,E1 -9444.388,E2 -9444.388} C_VEL
LIN {X 0,Y 431.147,Z 628.526,A -85,B 0,C 180,E1 -9446.262,E2 -9446.262} C_VEL
LIN {X 0,Y 431.199,Z 630.272,A -85,B 0,C 180,E1 -9448.132,E2 -9448.132} C_VEL
LIN {X 0,Y 431.164,Z 630.869,A -85,B 0,C 180,E1 -9450,E2 -9450} C_VEL
LIN {X 0,Y 431.199,Z 630.268,A -85,B 0,C 180,E1 -9451.868,E2 -9451.868} C_VEL
LIN {X 0,Y 431.147,Z 628.518,A -85,B 0,C 180,E1 -9453.738,E2 -9453.738} C_VEL
LIN {X 0,Y 431.213,Z 625.596,A -85,B 0,C 180,E1 -9455.612,E2 -9455.612} C_VEL
LIN {X 0,Y 431.345,Z 621.431,A -85,B 0,C 180,E1 -9457.489,E2 -9457.489} C_VEL
LIN {X 0,Y 431.589,Z 615.912,A -85,B 0,C 180,E1 -9459.372,E2 -9459.372} C_VEL
LIN {X 0,Y 432.094,Z 608.894,A -85,B 0,C 180,E1 -9461.255,E2 -9461.255} C_VEL
LIN {X 0,Y 432.663,Z 600.159,A -85,B 0,C 180,E1 -9463.144,E2 -9463.144} C_VEL
LIN {X 0,Y 433.433,Z 590.885,A -85,B 0,C 180,E1 -9464.796,E2 -9464.796} C_VEL
LIN {X 0,Y 434.254,Z 581.459,A -85,B 0,C 180,E1 -9466.21,E2 -9466.21} C_VEL
LIN {X 0,Y 435.288,Z 570.633,A -85,B 0,C 180,E1 -9467.576,E2 -9467.576} C_VEL
LIN {X 0,Y 436.385,Z 558.007,A -85,B 0,C 180,E1 -9468.911,E2 -9468.911} C_VEL
LIN {X 0,Y 437.633,Z 544.535,A -85,B 0,C 180,E1 -9470.075,E2 -9470.075} C_VEL
LIN {X 0,Y 438.714,Z 531.308,A -85,B 0,C 180,E1 -9471.004,E2 -9471.004} C_VEL
LIN {X 0,Y 439.672,Z 517.414,A -85,B 0,C 180,E1 -9471.785,E2 -9471.785} C_VEL
LIN {X 0,Y 440.526,Z 502.725,A -85,B 0,C 180,E1 -9472.416,E2 -9472.416} C_VEL
LIN {X 0,Y 441.171,Z 487.472,A -85,B 0,C 180,E1 -9472.879,E2 -9472.879} C_VEL
LIN {X 0,Y 441.638,Z 465.372,A -85,B 0,C 180,E1 -9473.287,E2 -9473.287} C_VEL
LIN {X 0,Y 443.405,Z 348.602,A -85,B 0,C 180,E1 -9475.218,E2 -9475.218} C_VEL
LIN {X 0,Y 437.469,Z 318.378,A -85,B 0,C 180,E1 -9476.12,E2 -9476.12} C_VEL
LIN {X 0,Y 438.105,Z 308.378,A -85,B 0,C 180,E1 -9477.723,E2 -9477.723} C_VEL
LIN {X 0,Y 435.791,Z 297.8,A -85,B 0,C 180,E1 -9479.648,E2 -9479.648} C_VEL
LIN {X 0,Y 432.313,Z 284.251,A -85,B 0,C 180,E1 -9482.237,E2 -9482.237} C_VEL
LIN {X 0,Y 432.334,Z 284.257,A -85,B 0,C 180,E1 -9484.676,E2 -9484.676} C_VEL
LIN {X 0,Y 432.317,Z 284.261,A -85,B 0,C 180,E1 -9488.151,E2 -9488.151} C_VEL
LIN {X 0,Y 432.297,Z 284.263,A -85,B 0,C 180,E1 -9491.8,E2 -9491.8} C_VEL
LIN {X 0,Y 432.325,Z 284.259,A -85,B 0,C 180,E1 -9494.347,E2 -9494.347} C_VEL
LIN {X 0,Y 432.299,Z 284.259,A -85,B 0,C 180,E1 -9497.017,E2 -9497.017} C_VEL
LIN {X 0,Y 432.28,Z 284.264,A -85,B 0,C 180,E1 -9499.827,E2 -9499.827} C_VEL
LIN {X 0,Y 432.286,Z 284.259,A -85,B 0,C 180,E1 -9503.02,E2 -9503.02} C_VEL
LIN {X 0,Y 432.323,Z 284.258,A -85,B 0,C 180,E1 -9506.001,E2 -9506.001} C_VEL
LIN {X 0,Y 432.336,Z 284.257,A -85,B 0,C 180,E1 -9509.49,E2 -9509.49} C_VEL
LIN {X 0,Y 432.324,Z 284.258,A -85,B 0,C 180,E1 -9511.873,E2 -9511.873} C_VEL
LIN {X 0,Y 432.337,Z 284.257,A -85,B 0,C 180,E1 -9515.547,E2 -9515.547} C_VEL
LIN {X 0,Y 432.338,Z 284.253,A -85,B 0,C 180,E1 -9519.046,E2 -9519.046} C_VEL
LIN {X 0,Y 432.345,Z 284.245,A -85,B 0,C 180,E1 -9522.01,E2 -9522.01} C_VEL
LIN {X 0,Y 432.378,Z 284.249,A -85,B 0,C 180,E1 -9524.926,E2 -9524.926} C_VEL
LIN {X 0,Y 432.44,Z 284.223,A -85,B 0,C 180,E1 -9527.803,E2 -9527.803} C_VEL
LIN {X 0,Y 432.433,Z 284.246,A -85,B 0,C 180,E1 -9531.589,E2 -9531.589} C_VEL
LIN {X 0,Y 432.57,Z 284.219,A -85,B 0,C 180,E1 -9534.406,E2 -9534.406} C_VEL
LIN {X 0,Y 432.582,Z 284.218,A -85,B 0,C 180,E1 -9538.138,E2 -9538.138} C_VEL
LIN {X 0,Y 432.588,Z 284.223,A -85,B 0,C 180,E1 -9540,E2 -9540} C_VEL
LIN {X 0,Y 432.557,Z 284.223,A -85,B 0,C 180,E1 -9542.794,E2 -9542.794} C_VEL
LIN {X 0,Y 432.571,Z 284.225,A -85,B 0,C 180,E1 -9545.594,E2 -9545.594} C_VEL
LIN {X 0,Y 432.451,Z 284.239,A -85,B 0,C 180,E1 -9548.411,E2 -9548.411} C_VEL
LIN {X 0,Y 432.446,Z 284.239,A -85,B 0,C 180,E1 -9552.197,E2 -9552.197} C_VEL
LIN {X 0,Y 432.418,Z 284.243,A -85,B 0,C 180,E1 -9556.039,E2 -9556.039} C_VEL
LIN {X 0,Y 432.376,Z 284.237,A -85,B 0,C 180,E1 -9559.485,E2 -9559.485} C_VEL
LIN {X 0,Y 432.306,Z 284.257,A -85,B 0,C 180,E1 -9562.965,E2 -9562.965} C_VEL
LIN {X 0,Y 432.34,Z 284.248,A -85,B 0,C 180,E1 -9566.034,E2 -9566.034} C_VEL
LIN {X 0,Y 432.333,Z 284.254,A -85,B 0,C 180,E1 -9569.188,E2 -9569.188} C_VEL
LIN {X 0,Y 432.312,Z 284.255,A -85,B 0,C 180,E1 -9572.444,E2 -9572.444} C_VEL
LIN {X 0,Y 432.329,Z 284.254,A -85,B 0,C 180,E1 -9575.819,E2 -9575.819} C_VEL
LIN {X 0,Y 432.321,Z 284.255,A -85,B 0,C 180,E1 -9579.346,E2 -9579.346} C_VEL
LIN {X 0,Y 432.327,Z 284.254,A -85,B 0,C 180,E1 -9581.798,E2 -9581.798} C_VEL
LIN {X 0,Y 432.328,Z 284.257,A -85,B 0,C 180,E1 -9584.348,E2 -9584.348} C_VEL
LIN {X 0,Y 432.315,Z 284.261,A -85,B 0,C 180,E1 -9587.017,E2 -9587.017} C_VEL
LIN {X 0,Y 432.336,Z 284.255,A -85,B 0,C 180,E1 -9589.821,E2 -9589.821} C_VEL
LIN {X 0,Y 432.303,Z 284.26,A -85,B 0,C 180,E1 -9593.023,E2 -9593.023} C_VEL
LIN {X 0,Y 432.354,Z 284.255,A -85,B 0,C 180,E1 -9595.998,E2 -9595.998} C_VEL
LIN {X 0,Y 432.345,Z 284.256,A -85,B 0,C 180,E1 -9599.491,E2 -9599.491} C_VEL
LIN {X 0,Y 432.37,Z 284.281,A -85,B 0,C 180,E1 -9601.218,E2 -9601.218} C_VEL
LIN {X 0,Y 435.346,Z 296.603,A -85,B 0,C 180,E1 -9603.799,E2 -9603.799} C_VEL
LIN {X 0,Y 441.537,Z 311.937,A -85,B 0,C 180,E1 -9604.47,E2 -9604.47} C_VEL
LIN {X 0,Y 443.758,Z 322.045,A -85,B 0,C 180,E1 -9604.785,E2 -9604.785} C_VEL
LIN {X 0,Y 441.948,Z 437.782,A -85,B 0,C 180,E1 -9606.699,E2 -9606.699} C_VEL
LIN {X 0,Y 441.49,Z 462.559,A -85,B 0,C 180,E1 -9607.138,E2 -9607.138} C_VEL
LIN {X 0,Y 440.932,Z 478.048,A -85,B 0,C 180,E1 -9607.595,E2 -9607.595} C_VEL
LIN {X 0,Y 440.302,Z 492.453,A -85,B 0,C 180,E1 -9608.205,E2 -9608.205} C_VEL
LIN {X 0,Y 439.291,Z 506.644,A -85,B 0,C 180,E1 -9608.987,E2 -9608.987} C_VEL
LIN {X 0,Y 438.286,Z 511.973,A -85,B 0,C 180,E1 -9609.3,E2 -9609.3} C_VEL
LIN {X 0,Y 434.921,Z 520.549,A -85,B 0,C 180,E1 -9609.791,E2 -9609.791} C_VEL
LIN {X 0,Y 431.491,Z 528.843,A -85,B 0,C 180,E1 -9610.351,E2 -9610.351} C_VEL
LIN {X 0,Y 430.384,Z 533.668,A -85,B 0,C 180,E1 -9610.767,E2 -9610.767} C_VEL
LIN {X 0,Y 429.333,Z 545.32,A -85,B 0,C 180,E1 -9612.003,E2 -9612.003} C_VEL
LIN {X 0,Y 428.241,Z 555.718,A -85,B 0,C 180,E1 -9613.31,E2 -9613.31} C_VEL
LIN {X 0,Y 427.313,Z 565.358,A -85,B 0,C 180,E1 -9614.743,E2 -9614.743} C_VEL
LIN {X 0,Y 426.308,Z 574.807,A -85,B 0,C 180,E1 -9616.413,E2 -9616.413} C_VEL
LIN {X 0,Y 425.718,Z 582.665,A -85,B 0,C 180,E1 -9618.091,E2 -9618.091} C_VEL
LIN {X 0,Y 425.011,Z 590.005,A -85,B 0,C 180,E1 -9620.001,E2 -9620.001} C_VEL
LIN {X 0,Y 424.644,Z 595.825,A -85,B 0,C 180,E1 -9621.913,E2 -9621.913} C_VEL
LIN {X 0,Y 424.448,Z 599.513,A -85,B 0,C 180,E1 -9623.454,E2 -9623.454} C_VEL
LIN {X 0,Y 424.222,Z 602.765,A -85,B 0,C 180,E1 -9625.249,E2 -9625.249} C_VEL
LIN {X 0,Y 424.222,Z 605.073,A -85,B 0,C 180,E1 -9627.151,E2 -9627.151} C_VEL
LIN {X 0,Y 424.089,Z 606.257,A -85,B 0,C 180,E1 -9629.05,E2 -9629.05} C_VEL
LIN {X 0,Y 424.089,Z 606.273,A -85,B 0,C 180,E1 -9630.95,E2 -9630.95} C_VEL
LIN {X 0,Y 424.219,Z 605.155,A -85,B 0,C 180,E1 -9632.849,E2 -9632.849} C_VEL
LIN {X 0,Y 424.219,Z 602.911,A -85,B 0,C 180,E1 -9634.751,E2 -9634.751} C_VEL
LIN {X 0,Y 424.421,Z 599.477,A -85,B 0,C 180,E1 -9636.656,E2 -9636.656} C_VEL
LIN {X 0,Y 424.715,Z 594.777,A -85,B 0,C 180,E1 -9638.565,E2 -9638.565} C_VEL
LIN {X 0,Y 425.094,Z 588.688,A -85,B 0,C 180,E1 -9640.478,E2 -9640.478} C_VEL
LIN {X 0,Y 425.833,Z 581.013,A -85,B 0,C 180,E1 -9642.389,E2 -9642.389} C_VEL
LIN {X 0,Y 426.523,Z 572.832,A -85,B 0,C 180,E1 -9644.066,E2 -9644.066} C_VEL
LIN {X 0,Y 427.511,Z 562.972,A -85,B 0,C 180,E1 -9645.738,E2 -9645.738} C_VEL
LIN {X 0,Y 428.508,Z 552.86,A -85,B 0,C 180,E1 -9647.17,E2 -9647.17} C_VEL
LIN {X 0,Y 429.676,Z 541.198,A -85,B 0,C 180,E1 -9648.555,E2 -9648.555} C_VEL
LIN {X 0,Y 430.888,Z 528.738,A -85,B 0,C 180,E1 -9649.781,E2 -9649.781} C_VEL
LIN {X 0,Y 432.015,Z 515.612,A -85,B 0,C 180,E1 -9650.846,E2 -9650.846} C_VEL
LIN {X 0,Y 432.983,Z 503.105,A -85,B 0,C 180,E1 -9651.67,E2 -9651.67} C_VEL
LIN {X 0,Y 433.864,Z 489.381,A -85,B 0,C 180,E1 -9652.393,E2 -9652.393} C_VEL
LIN {X 0,Y 434.544,Z 475.092,A -85,B 0,C 180,E1 -9652.965,E2 -9652.965} C_VEL
LIN {X 0,Y 435.059,Z 460.176,A -85,B 0,C 180,E1 -9653.377,E2 -9653.377} C_VEL
LIN {X 0,Y 436.355,Z 382.684,A -85,B 0,C 180,E1 -9654.692,E2 -9654.692} C_VEL
LIN {X 0,Y 437.251,Z 322.44,A -85,B 0,C 180,E1 -9655.71,E2 -9655.71} C_VEL
LIN {X 0,Y 434.735,Z 312.252,A -85,B 0,C 180,E1 -9656.055,E2 -9656.055} C_VEL
LIN {X 0,Y 428.139,Z 296.782,A -85,B 0,C 180,E1 -9656.776,E2 -9656.776} C_VEL
LIN {X 0,Y 425.302,Z 285.135,A -85,B 0,C 180,E1 -9659.306,E2 -9659.306} C_VEL
LIN {X 0,Y 425.279,Z 285.137,A -85,B 0,C 180,E1 -9662.562,E2 -9662.562} C_VEL
LIN {X 0,Y 425.297,Z 285.137,A -85,B 0,C 180,E1 -9665.335,E2 -9665.335} C_VEL
LIN {X 0,Y 425.301,Z 285.137,A -85,B 0,C 180,E1 -9668.897,E2 -9668.897} C_VEL
LIN {X 0,Y 425.285,Z 285.135,A -85,B 0,C 180,E1 -9671.957,E2 -9671.957} C_VEL
LIN {X 0,Y 425.279,Z 285.137,A -85,B 0,C 180,E1 -9675.282,E2 -9675.282} C_VEL
LIN {X 0,Y 425.26,Z 285.125,A -85,B 0,C 180,E1 -9678.62,E2 -9678.62} C_VEL
LIN {X 0,Y 425.285,Z 285.137,A -85,B 0,C 180,E1 -9681.1,E2 -9681.1} C_VEL
LIN {X 0,Y 425.287,Z 285.126,A -85,B 0,C 180,E1 -9684.663,E2 -9684.663} C_VEL
LIN {X 0,Y 425.254,Z 285.129,A -85,B 0,C 180,E1 -9688.072,E2 -9688.072} C_VEL
LIN {X 0,Y 425.322,Z 285.129,A -85,B 0,C 180,E1 -9691.367,E2 -9691.367} C_VEL
LIN {X 0,Y 425.273,Z 285.133,A -85,B 0,C 180,E1 -9694.553,E2 -9694.553} C_VEL
LIN {X 0,Y 425.273,Z 285.136,A -85,B 0,C 180,E1 -9696.633,E2 -9696.633} C_VEL
LIN {X 0,Y 425.284,Z 285.132,A -85,B 0,C 180,E1 -9699.694,E2 -9699.694} C_VEL
LIN {X 0,Y 425.322,Z 285.126,A -85,B 0,C 180,E1 -9702.696,E2 -9702.696} C_VEL
LIN {X 0,Y 425.334,Z 285.123,A -85,B 0,C 180,E1 -9705.649,E2 -9705.649} C_VEL
LIN {X 0,Y 425.335,Z 285.128,A -85,B 0,C 180,E1 -9708.563,E2 -9708.563} C_VEL
LIN {X 0,Y 425.494,Z 285.105,A -85,B 0,C 180,E1 -9712.31,E2 -9712.31} C_VEL
LIN {X 0,Y 425.528,Z 285.104,A -85,B 0,C 180,E1 -9714.313,E2 -9714.313} C_VEL
LIN {X 0,Y 425.559,Z 285.099,A -85,B 0,C 180,E1 -9718.107,E2 -9718.107} C_VEL
LIN {X 0,Y 425.682,Z 285.079,A -85,B 0,C 180,E1 -9720,E2 -9720} C_VEL
LIN {X 0,Y 425.506,Z 285.107,A -85,B 0,C 180,E1 -9722.84,E2 -9722.84} C_VEL
LIN {X 0,Y 425.527,Z 285.099,A -85,B 0,C 180,E1 -9725.687,E2 -9725.687} C_VEL
LIN {X 0,Y 425.392,Z 285.119,A -85,B 0,C 180,E1 -9728.551,E2 -9728.551} C_VEL
LIN {X 0,Y 425.399,Z 285.122,A -85,B 0,C 180,E1 -9732.402,E2 -9732.402} C_VEL
LIN {X 0,Y 425.374,Z 285.128,A -85,B 0,C 180,E1 -9736.312,E2 -9736.312} C_VEL
LIN {X 0,Y 425.317,Z 285.13,A -85,B 0,C 180,E1 -9739.636,E2 -9739.636} C_VEL
LIN {X 0,Y 425.276,Z 285.134,A -85,B 0,C 180,E1 -9742.339,E2 -9742.339} C_VEL
LIN {X 0,Y 425.246,Z 285.135,A -85,B 0,C 180,E1 -9745.448,E2 -9745.448} C_VEL
LIN {X 0,Y 425.303,Z 285.131,A -85,B 0,C 180,E1 -9748.862,E2 -9748.862} C_VEL
LIN {X 0,Y 425.254,Z 285.14,A -85,B 0,C 180,E1 -9751.928,E2 -9751.928} C_VEL
LIN {X 0,Y 425.282,Z 285.133,A -85,B 0,C 180,E1 -9755.337,E2 -9755.337} C_VEL
LIN {X 0,Y 425.267,Z 285.132,A -85,B 0,C 180,E1 -9758.902,E2 -9758.902} C_VEL
LIN {X 0,Y 425.253,Z 285.138,A -85,B 0,C 180,E1 -9762.656,E2 -9762.656} C_VEL
LIN {X 0,Y 425.276,Z 285.135,A -85,B 0,C 180,E1 -9765.284,E2 -9765.284} C_VEL
LIN {X 0,Y 425.241,Z 285.139,A -85,B 0,C 180,E1 -9768.619,E2 -9768.619} C_VEL
LIN {X 0,Y 425.27,Z 285.134,A -85,B 0,C 180,E1 -9771.1,E2 -9771.1} C_VEL
LIN {X 0,Y 425.293,Z 285.135,A -85,B 0,C 180,E1 -9774.665,E2 -9774.665} C_VEL
LIN {X 0,Y 425.317,Z 285.32,A -85,B 0,C 180,E1 -9777.385,E2 -9777.385} C_VEL
LIN {X 0,Y 428.665,Z 298.377,A -85,B 0,C 180,E1 -9779.937,E2 -9779.937} C_VEL
LIN {X 0,Y 431.317,Z 310.257,A -85,B 0,C 180,E1 -9782.147,E2 -9782.147} C_VEL
LIN {X 0,Y 430.783,Z 318.259,A -85,B 0,C 180,E1 -9783.438,E2 -9783.438} C_VEL
LIN {X 0,Y 436.929,Z 349.226,A -85,B 0,C 180,E1 -9784.391,E2 -9784.391} C_VEL
LIN {X 0,Y 435.3,Z 456.522,A -85,B 0,C 180,E1 -9786.195,E2 -9786.195} C_VEL
LIN {X 0,Y 434.676,Z 486.311,A -85,B 0,C 180,E1 -9786.728,E2 -9786.728} C_VEL
LIN {X 0,Y 434.011,Z 501.938,A -85,B 0,C 180,E1 -9787.2,E2 -9787.2} C_VEL
LIN {X 0,Y 433.097,Z 516.461,A -85,B 0,C 180,E1 -9787.82,E2 -9787.82} C_VEL
LIN {X 0,Y 432.222,Z 529.37,A -85,B 0,C 180,E1 -9788.541,E2 -9788.541} C_VEL
LIN {X 0,Y 431.051,Z 542.87,A -85,B 0,C 180,E1 -9789.48,E2 -9789.48} C_VEL
LIN {X 0,Y 429.75,Z 556.619,A -85,B 0,C 180,E1 -9790.661,E2 -9790.661} C_VEL
LIN {X 0,Y 428.475,Z 569.791,A -85,B 0,C 180,E1 -9792.052,E2 -9792.052} C_VEL
LIN {X 0,Y 427.364,Z 581.282,A -85,B 0,C 180,E1 -9793.521,E2 -9793.521} C_VEL
LIN {X 0,Y 426.357,Z 592.146,A -85,B 0,C 180,E1 -9795.197,E2 -9795.197} C_VEL
LIN {X 0,Y 425.467,Z 601.591,A -85,B 0,C 180,E1 -9796.958,E2 -9796.958} C_VEL
LIN {X 0,Y 425.084,Z 608.71,A -85,B 0,C 180,E1 -9798.557,E2 -9798.557} C_VEL
LIN {X 0,Y 424.523,Z 615.717,A -85,B 0,C 180,E1 -9800.471,E2 -9800.471} C_VEL
LIN {X 0,Y 424.307,Z 621.232,A -85,B 0,C 180,E1 -9802.386,E2 -9802.386} C_VEL
LIN {X 0,Y 424.138,Z 625.4,A -85,B 0,C 180,E1 -9804.294,E2 -9804.294} C_VEL
LIN {X 0,Y 424.059,Z 628.324,A -85,B 0,C 180,E1 -9806.199,E2 -9806.199} C_VEL
LIN {X 0,Y 424.125,Z 630.07,A -85,B 0,C 180,E1 -9808.101,E2 -9808.101} C_VEL
LIN {X 0,Y 424.081,Z 630.666,A -85,B 0,C 180,E1 -9810,E2 -9810} C_VEL
LIN {X 0,Y 424.125,Z 630.066,A -85,B 0,C 180,E1 -9811.899,E2 -9811.899} C_VEL
LIN {X 0,Y 424.059,Z 628.315,A -85,B 0,C 180,E1 -9813.801,E2 -9813.801} C_VEL
LIN {X 0,Y 424.126,Z 625.392,A -85,B 0,C 180,E1 -9815.706,E2 -9815.706} C_VEL
LIN {X 0,Y 424.282,Z 621.226,A -85,B 0,C 180,E1 -9817.615,E2 -9817.615} C_VEL
LIN {X 0,Y 424.523,Z 615.706,A -85,B 0,C 180,E1 -9819.529,E2 -9819.529} C_VEL
LIN {X 0,Y 425.079,Z 608.688,A -85,B 0,C 180,E1 -9821.443,E2 -9821.443} C_VEL
LIN {X 0,Y 425.675,Z 599.952,A -85,B 0,C 180,E1 -9823.364,E2 -9823.364} C_VEL
LIN {X 0,Y 426.485,Z 590.678,A -85,B 0,C 180,E1 -9825.042,E2 -9825.042} C_VEL
LIN {X 0,Y 427.389,Z 581.252,A -85,B 0,C 180,E1 -9826.478,E2 -9826.478} C_VEL
LIN {X 0,Y 428.554,Z 569.464,A -85,B 0,C 180,E1 -9827.981,E2 -9827.981} C_VEL
LIN {X 0,Y 429.75,Z 556.578,A -85,B 0,C 180,E1 -9829.339,E2 -9829.339} C_VEL
LIN {X 0,Y 431.046,Z 542.803,A -85,B 0,C 180,E1 -9830.52,E2 -9830.52} C_VEL
LIN {X 0,Y 432.206,Z 529.279,A -85,B 0,C 180,E1 -9831.46,E2 -9831.46} C_VEL
LIN {X 0,Y 433.214,Z 515.324,A -85,B 0,C 180,E1 -9832.231,E2 -9832.231} C_VEL
LIN {X 0,Y 434.076,Z 500.134,A -85,B 0,C 180,E1 -9832.865,E2 -9832.865} C_VEL
LIN {X 0,Y 434.736,Z 484.971,A -85,B 0,C 180,E1 -9833.301,E2 -9833.301} C_VEL
LIN {X 0,Y 436.856,Z 361.138,A -85,B 0,C 180,E1 -9835.396,E2 -9835.396} C_VEL
LIN {X 0,Y 436.908,Z 349.278,A -85,B 0,C 180,E1 -9835.604,E2 -9835.604} C_VEL
LIN {X 0,Y 430.777,Z 318.06,A -85,B 0,C 180,E1 -9836.565,E2 -9836.565} C_VEL
LIN {X 0,Y 431.316,Z 310.21,A -85,B 0,C 180,E1 -9837.854,E2 -9837.854} C_VEL
LIN {X 0,Y 428.663,Z 298.323,A -85,B 0,C 180,E1 -9840.064,E2 -9840.064} C_VEL
LIN {X 0,Y 425.286,Z 285.128,A -85,B 0,C 180,E1 -9842.654,E2 -9842.654} C_VEL
LIN {X 0,Y 425.274,Z 285.139,A -85,B 0,C 180,E1 -9845.927,E2 -9845.927} C_VEL
LIN {X 0,Y 425.252,Z 285.139,A -85,B 0,C 180,E1 -9849.036,E2 -9849.036} C_VEL
LIN {X 0,Y 425.25,Z 285.139,A -85,B 0,C 180,E1 -9852.655,E2 -9852.655} C_VEL
LIN {X 0,Y 425.276,Z 285.135,A -85,B 0,C 180,E1 -9855.283,E2 -9855.283} C_VEL
LIN {X 0,Y 425.243,Z 285.139,A -85,B 0,C 180,E1 -9858.618,E2 -9858.618} C_VEL
LIN {X 0,Y 425.267,Z 285.135,A -85,B 0,C 180,E1 -9861.098,E2 -9861.098} C_VEL
LIN {X 0,Y 425.283,Z 285.13,A -85,B 0,C 180,E1 -9864.663,E2 -9864.663} C_VEL
LIN {X 0,Y 425.253,Z 285.139,A -85,B 0,C 180,E1 -9868.072,E2 -9868.072} C_VEL
LIN {X 0,Y 425.296,Z 285.132,A -85,B 0,C 180,E1 -9871.365,E2 -9871.365} C_VEL
LIN {X 0,Y 425.246,Z 285.137,A -85,B 0,C 180,E1 -9874.552,E2 -9874.552} C_VEL
LIN {X 0,Y 425.281,Z 285.138,A -85,B 0,C 180,E1 -9877.729,E2 -9877.729} C_VEL
LIN {X 0,Y 425.349,Z 285.11,A -85,B 0,C 180,E1 -9880.704,E2 -9880.704} C_VEL
LIN {X 0,Y 425.375,Z 285.123,A -85,B 0,C 180,E1 -9883.688,E2 -9883.688} C_VEL
LIN {X 0,Y 425.396,Z 285.102,A -85,B 0,C 180,E1 -9887.598,E2 -9887.598} C_VEL
LIN {X 0,Y 425.381,Z 285.122,A -85,B 0,C 180,E1 -9891.449,E2 -9891.449} C_VEL
LIN {X 0,Y 425.526,Z 285.096,A -85,B 0,C 180,E1 -9894.313,E2 -9894.313} C_VEL
LIN {X 0,Y 425.551,Z 285.094,A -85,B 0,C 180,E1 -9898.107,E2 -9898.107} C_VEL
LIN {X 0,Y 425.424,Z 285.117,A -85,B 0,C 180,E1 -9900.947,E2 -9900.947} C_VEL
LIN {X 0,Y 425.512,Z 285.101,A -85,B 0,C 180,E1 -9902.84,E2 -9902.84} C_VEL
LIN {X 0,Y 425.492,Z 285.104,A -85,B 0,C 180,E1 -9906.592,E2 -9906.592} C_VEL
LIN {X 0,Y 425.384,Z 285.121,A -85,B 0,C 180,E1 -9909.51,E2 -9909.51} C_VEL
LIN {X 0,Y 425.382,Z 285.123,A -85,B 0,C 180,E1 -9912.904,E2 -9912.904} C_VEL
LIN {X 0,Y 425.35,Z 285.125,A -85,B 0,C 180,E1 -9916.605,E2 -9916.605} C_VEL
LIN {X 0,Y 425.317,Z 285.114,A -85,B 0,C 180,E1 -9919.636,E2 -9919.636} C_VEL
LIN {X 0,Y 425.293,Z 285.135,A -85,B 0,C 180,E1 -9923.366,E2 -9923.366} C_VEL
LIN {X 0,Y 425.331,Z 285.117,A -85,B 0,C 180,E1 -9926.843,E2 -9926.843} C_VEL
LIN {X 0,Y 425.281,Z 285.132,A -85,B 0,C 180,E1 -9929.72,E2 -9929.72} C_VEL
LIN {X 0,Y 425.261,Z 285.14,A -85,B 0,C 180,E1 -9933.05,E2 -9933.05} C_VEL
LIN {X 0,Y 425.273,Z 285.133,A -85,B 0,C 180,E1 -9935.929,E2 -9935.929} C_VEL
LIN {X 0,Y 425.275,Z 285.136,A -85,B 0,C 180,E1 -9939.042,E2 -9939.042} C_VEL
LIN {X 0,Y 425.283,Z 285.132,A -85,B 0,C 180,E1 -9941.959,E2 -9941.959} C_VEL
LIN {X 0,Y 425.279,Z 285.135,A -85,B 0,C 180,E1 -9945.284,E2 -9945.284} C_VEL
LIN {X 0,Y 425.27,Z 285.138,A -85,B 0,C 180,E1 -9948.622,E2 -9948.622} C_VEL
LIN {X 0,Y 425.308,Z 285.126,A -85,B 0,C 180,E1 -9951.104,E2 -9951.104} C_VEL
LIN {X 0,Y 425.294,Z 285.131,A -85,B 0,C 180,E1 -9954.665,E2 -9954.665} C_VEL
LIN {X 0,Y 425.262,Z 285.14,A -85,B 0,C 180,E1 -9958.074,E2 -9958.074} C_VEL
LIN {X 0,Y 425.32,Z 285.239,A -85,B 0,C 180,E1 -9960.845,E2 -9960.845} C_VEL
LIN {X 0,Y 428.212,Z 296.865,A -85,B 0,C 180,E1 -9963.329,E2 -9963.329} C_VEL
LIN {X 0,Y 435.311,Z 313.944,A -85,B 0,C 180,E1 -9964.11,E2 -9964.11} C_VEL
LIN {X 0,Y 437.356,Z 322.989,A -85,B 0,C 180,E1 -9964.403,E2 -9964.403} C_VEL
LIN {X 0,Y 435.091,Z 458.614,A -85,B 0,C 180,E1 -9966.688,E2 -9966.688} C_VEL
LIN {X 0,Y 434.584,Z 473.24,A -85,B 0,C 180,E1 -9967.069,E2 -9967.069} C_VEL
LIN {X 0,Y 433.929,Z 487.89,A -85,B 0,C 180,E1 -9967.634,E2 -9967.634} C_VEL
LIN {X 0,Y 433.079,Z 501.588,A -85,B 0,C 180,E1 -9968.335,E2 -9968.335} C_VEL
LIN {X 0,Y 432.078,Z 514.399,A -85,B 0,C 180,E1 -9969.158,E2 -9969.158} C_VEL
LIN {X 0,Y 430.96,Z 527.757,A -85,B 0,C 180,E1 -9970.222,E2 -9970.222} C_VEL
LIN {X 0,Y 430.384,Z 533.668,A -85,B 0,C 180,E1 -9970.767,E2 -9970.767} C_VEL
LIN {X 0,Y 429.269,Z 538.461,A -85,B 0,C 180,E1 -9971.209,E2 -9971.209} C_VEL
LIN {X 0,Y 425.761,Z 546.095,A -85,B 0,C 180,E1 -9971.925,E2 -9971.925} C_VEL
LIN {X 0,Y 422.305,Z 553.361,A -85,B 0,C 180,E1 -9972.708,E2 -9972.708} C_VEL
LIN {X 0,Y 421.269,Z 557.507,A -85,B 0,C 180,E1 -9973.249,E2 -9973.249} C_VEL
LIN {X 0,Y 420.095,Z 568.492,A -85,B 0,C 180,E1 -9974.971,E2 -9974.971} C_VEL
LIN {X 0,Y 419.055,Z 577.861,A -85,B 0,C 180,E1 -9976.756,E2 -9976.756} C_VEL
LIN {X 0,Y 418.52,Z 584.871,A -85,B 0,C 180,E1 -9978.375,E2 -9978.375} C_VEL
LIN {X 0,Y 417.884,Z 591.809,A -85,B 0,C 180,E1 -9980.318,E2 -9980.318} C_VEL
LIN {X 0,Y 417.513,Z 597.259,A -85,B 0,C 180,E1 -9982.261,E2 -9982.261} C_VEL
LIN {X 0,Y 417.277,Z 601.374,A -85,B 0,C 180,E1 -9984.2,E2 -9984.2} C_VEL
LIN {X 0,Y 417.075,Z 604.268,A -85,B 0,C 180,E1 -9986.135,E2 -9986.135} C_VEL
LIN {X 0,Y 417.078,Z 606.006,A -85,B 0,C 180,E1 -9988.069,E2 -9988.069} C_VEL
LIN {X 0,Y 417.002,Z 606.617,A -85,B 0,C 180,E1 -9990,E2 -9990} C_VEL
LIN {X 0,Y 417.078,Z 606.055,A -85,B 0,C 180,E1 -9991.931,E2 -9991.931} C_VEL
LIN {X 0,Y 417.065,Z 604.381,A -85,B 0,C 180,E1 -9993.865,E2 -9993.865} C_VEL
LIN {X 0,Y 417.264,Z 601.548,A -85,B 0,C 180,E1 -9995.8,E2 -9995.8} C_VEL
LIN {X 0,Y 417.479,Z 597.495,A -85,B 0,C 180,E1 -9997.74,E2 -9997.74} C_VEL
LIN {X 0,Y 417.871,Z 592.118,A -85,B 0,C 180,E1 -9999.682,E2 -9999.682} C_VEL
LIN {X 0,Y 418.506,Z 585.263,A -85,B 0,C 180,E1 -10001.625,E2 -10001.625} C_VEL
LIN {X 0,Y 419.236,Z 576.708,A -85,B 0,C 180,E1 -10003.573,E2 -10003.573} C_VEL
LIN {X 0,Y 420.203,Z 567.607,A -85,B 0,C 180,E1 -10005.273,E2 -10005.273} C_VEL
LIN {X 0,Y 421.191,Z 558.329,A -85,B 0,C 180,E1 -10006.728,E2 -10006.728} C_VEL
LIN {X 0,Y 422.367,Z 547.312,A -85,B 0,C 180,E1 -10008.179,E2 -10008.179} C_VEL
LIN {X 0,Y 423.531,Z 535.244,A -85,B 0,C 180,E1 -10009.508,E2 -10009.508} C_VEL
LIN {X 0,Y 424.887,Z 521.984,A -85,B 0,C 180,E1 -10010.705,E2 -10010.705} C_VEL
LIN {X 0,Y 425.952,Z 508.985,A -85,B 0,C 180,E1 -10011.664,E2 -10011.664} C_VEL
LIN {X 0,Y 427.019,Z 495.487,A -85,B 0,C 180,E1 -10012.457,E2 -10012.457} C_VEL
LIN {X 0,Y 427.732,Z 480.862,A -85,B 0,C 180,E1 -10013.132,E2 -10013.132} C_VEL
LIN {X 0,Y 428.373,Z 465.286,A -85,B 0,C 180,E1 -10013.636,E2 -10013.636} C_VEL
LIN {X 0,Y 428.868,Z 445.405,A -85,B 0,C 180,E1 -10014.023,E2 -10014.023} C_VEL
LIN {X 0,Y 429.938,Z 381.074,A -85,B 0,C 180,E1 -10015.118,E2 -10015.118} C_VEL
LIN {X 0,Y 430.852,Z 323.54,A -85,B 0,C 180,E1 -10016.104,E2 -10016.104} C_VEL
LIN {X 0,Y 428.619,Z 314.715,A -85,B 0,C 180,E1 -10016.413,E2 -10016.413} C_VEL
LIN {X 0,Y 420.934,Z 296.9,A -85,B 0,C 180,E1 -10017.292,E2 -10017.292} C_VEL
LIN {X 0,Y 418.265,Z 286.013,A -85,B 0,C 180,E1 -10019.713,E2 -10019.713} C_VEL
LIN {X 0,Y 418.246,Z 286.017,A -85,B 0,C 180,E1 -10023.676,E2 -10023.676} C_VEL
LIN {X 0,Y 418.24,Z 286.012,A -85,B 0,C 180,E1 -10027.223,E2 -10027.223} C_VEL
LIN {X 0,Y 418.243,Z 286.008,A -85,B 0,C 180,E1 -10029.681,E2 -10029.681} C_VEL
LIN {X 0,Y 418.225,Z 286.014,A -85,B 0,C 180,E1 -10032.32,E2 -10032.32} C_VEL
LIN {X 0,Y 418.23,Z 286.014,A -85,B 0,C 180,E1 -10035.108,E2 -10035.108} C_VEL
LIN {X 0,Y 418.228,Z 286.001,A -85,B 0,C 180,E1 -10037.765,E2 -10037.765} C_VEL
LIN {X 0,Y 418.235,Z 286.012,A -85,B 0,C 180,E1 -10040.62,E2 -10040.62} C_VEL
LIN {X 0,Y 418.234,Z 286.003,A -85,B 0,C 180,E1 -10043.975,E2 -10043.975} C_VEL
LIN {X 0,Y 418.234,Z 286.007,A -85,B 0,C 180,E1 -10047.471,E2 -10047.471} C_VEL
LIN {X 0,Y 418.26,Z 286,A -85,B 0,C 180,E1 -10050.895,E2 -10050.895} C_VEL
LIN {X 0,Y 418.251,Z 286.005,A -85,B 0,C 180,E1 -10054.095,E2 -10054.095} C_VEL
LIN {X 0,Y 418.221,Z 286.012,A -85,B 0,C 180,E1 -10057.263,E2 -10057.263} C_VEL
LIN {X 0,Y 418.272,Z 286.007,A -85,B 0,C 180,E1 -10060.364,E2 -10060.364} C_VEL
LIN {X 0,Y 418.305,Z 286.003,A -85,B 0,C 180,E1 -10063.404,E2 -10063.404} C_VEL
LIN {X 0,Y 418.335,Z 285.997,A -85,B 0,C 180,E1 -10066.999,E2 -10066.999} C_VEL
LIN {X 0,Y 418.325,Z 286,A -85,B 0,C 180,E1 -10070.328,E2 -10070.328} C_VEL
LIN {X 0,Y 418.456,Z 285.984,A -85,B 0,C 180,E1 -10073.248,E2 -10073.248} C_VEL
LIN {X 0,Y 418.316,Z 285.995,A -85,B 0,C 180,E1 -10075.181,E2 -10075.181} C_VEL
LIN {X 0,Y 418.528,Z 285.975,A -85,B 0,C 180,E1 -10078.075,E2 -10078.075} C_VEL
LIN {X 0,Y 418.652,Z 285.954,A -85,B 0,C 180,E1 -10080,E2 -10080} C_VEL
LIN {X 0,Y 418.463,Z 285.984,A -85,B 0,C 180,E1 -10082.888,E2 -10082.888} C_VEL
LIN {X 0,Y 418.486,Z 285.977,A -85,B 0,C 180,E1 -10085.783,E2 -10085.783} C_VEL
LIN {X 0,Y 418.362,Z 285.993,A -85,B 0,C 180,E1 -10088.696,E2 -10088.696} C_VEL
LIN {X 0,Y 418.298,Z 286.003,A -85,B 0,C 180,E1 -10091.631,E2 -10091.631} C_VEL
LIN {X 0,Y 418.287,Z 286.007,A -85,B 0,C 180,E1 -10094.597,E2 -10094.597} C_VEL
LIN {X 0,Y 418.266,Z 286.004,A -85,B 0,C 180,E1 -10097.605,E2 -10097.605} C_VEL
LIN {X 0,Y 418.238,Z 286.012,A -85,B 0,C 180,E1 -10100.663,E2 -10100.663} C_VEL
LIN {X 0,Y 418.244,Z 286.011,A -85,B 0,C 180,E1 -10103.784,E2 -10103.784} C_VEL
LIN {X 0,Y 418.205,Z 286.015,A -85,B 0,C 180,E1 -10107.045,E2 -10107.045} C_VEL
LIN {X 0,Y 418.232,Z 286.015,A -85,B 0,C 180,E1 -10110.273,E2 -10110.273} C_VEL
LIN {X 0,Y 418.222,Z 286.008,A -85,B 0,C 180,E1 -10113.679,E2 -10113.679} C_VEL
LIN {X 0,Y 418.223,Z 286.011,A -85,B 0,C 180,E1 -10117.226,E2 -10117.226} C_VEL
LIN {X 0,Y 418.2,Z 286.002,A -85,B 0,C 180,E1 -10120.868,E2 -10120.868} C_VEL
LIN {X 0,Y 418.197,Z 286.019,A -85,B 0,C 180,E1 -10123.729,E2 -10123.729} C_VEL
LIN {X 0,Y 418.192,Z 286.017,A -85,B 0,C 180,E1 -10126.448,E2 -10126.448} C_VEL
LIN {X 0,Y 418.2,Z 286.015,A -85,B 0,C 180,E1 -10129.134,E2 -10129.134} C_VEL
LIN {X 0,Y 418.229,Z 286.011,A -85,B 0,C 180,E1 -10132.776,E2 -10132.776} C_VEL
